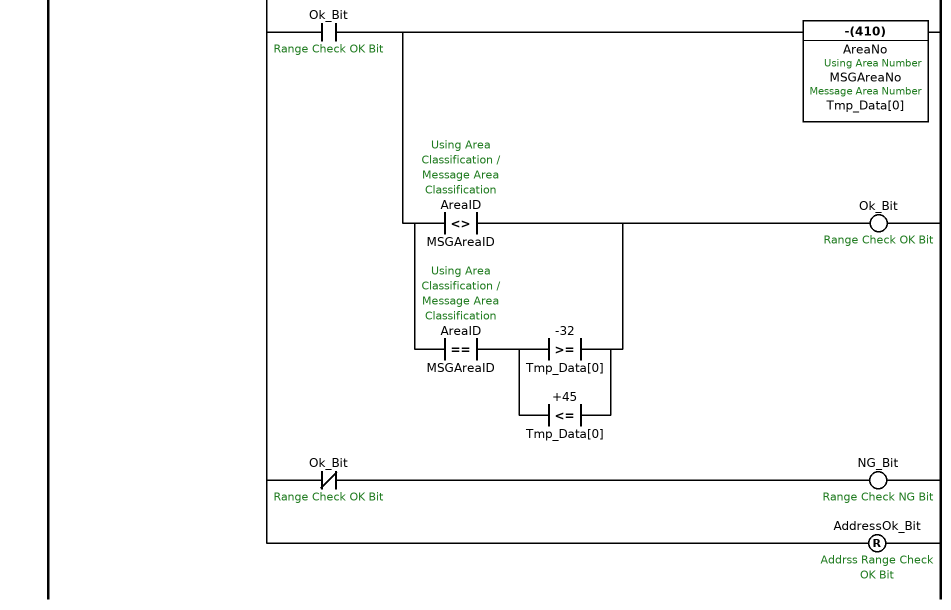
; [picture p24: FB INV002_Refresh_X31_, rungs 2-2]
; rung 2: Check input data range
LD EN
ANDNOT BUSY_Run  ; Internal Processing Flag
OR Data_Change  ; Detect input data change
OUT TR0
LD>=(325) &15 UnitSelect  ; Specify the connetcted Unit SCB=#BBBB_SCU=&0to&15
OR=(300) #BBBB UnitSelect  ; Specify the connetcted Unit SCB=#BBBB_SCU=&0to&15
OR=(300) #CCCC UnitSelect  ; Specify the connetcted Unit SCB=#BBBB_SCU=&0to&15
ANDLD
OUT Ok_Bit  ; Range Check OK Bit
LD TR0
AND Ok_Bit  ; Range Check OK Bit
AND<=(315) &1 PortNo  ; Serial port No. &0to&2
AND>=(325) &2 PortNo  ; Serial port No. &0to&2
OUT Ok_Bit  ; Range Check OK Bit
LD TR0
+(400) #4F P_EM_MaxNo EM_NoCheck  ; EM bank size, EM bank size check area
MOV(021) &62 Tmp_Data[0]
AND Ok_Bit  ; Range Check OK Bit
OUT TR1
AND=(300) #B0 AreaID  ; Using Area Classification
-(410) &6144 Tmp_Data[0] Tmp_Data[1]
AND>(320) Tmp_Data[1] AreaNo  ; Using Area Number
OUT Ok_IO  ; Selected CIO area range OK
LD TR1
AND=(300) #B1 AreaID  ; Using Area Classification
-(410) &512 Tmp_Data[0] Tmp_Data[1]
AND>(320) Tmp_Data[1] AreaNo  ; Using Area Number
OUT Ok_WR  ; Selected WR area range OK
LD TR1
AND=(300) #B2 AreaID  ; Using Area Classification
-(410) &512 Tmp_Data[0] Tmp_Data[1]
AND>(320) Tmp_Data[1] AreaNo  ; Using Area Number
OUT Ok_HR  ; Selected HR area range OK
LD TR1
AND=(300) #82 AreaID  ; Using Area Classification
-(410) &32768 Tmp_Data[0] Tmp_Data[1]
AND>(320) Tmp_Data[1] AreaNo  ; Using Area Number
OUT Ok_DM  ; Selected DM area range OK
LD TR1
AND<=(315) #50 AreaID  ; Using Area Classification
AND>=(325) EM_NoCheck AreaID  ; EM bank size check area, Using Area Classification
-(410) &32768 Tmp_Data[0] Tmp_Data[1]
AND>(320) Tmp_Data[1] AreaNo  ; Using Area Number
OUT Ok_EM  ; Selected EM area range OK
LD TR0
LD Ok_IO  ; Selected CIO area range OK
OR Ok_WR  ; Selected WR area range OK
OR Ok_HR  ; Selected HR area range OK
OR Ok_DM  ; Selected DM area range OK
OR Ok_EM  ; Selected EM area range OK
ANDLD
OUT Ok_Bit  ; Range Check OK Bit
LD TR0
MOV(021) &45 Tmp_Data[0]
AND Ok_Bit  ; Range Check OK Bit
OUT TR2
AND=(300) #B0 MSGAreaID  ; Message Area Classification
-(410) &6144 Tmp_Data[0] Tmp_Data[1]
AND>(320) Tmp_Data[1] MSGAreaNo  ; Message Area Number
OUT Ok_IO  ; Selected CIO area range OK
LD TR2
AND=(300) #B1 MSGAreaID  ; Message Area Classification
-(410) &512 Tmp_Data[0] Tmp_Data[1]
AND>(320) Tmp_Data[1] MSGAreaNo  ; Message Area Number
OUT Ok_WR  ; Selected WR area range OK
LD TR2
AND=(300) #B2 MSGAreaID  ; Message Area Classification
-(410) &512 Tmp_Data[0] Tmp_Data[1]
AND>(320) Tmp_Data[1] MSGAreaNo  ; Message Area Number
OUT Ok_HR  ; Selected HR area range OK
LD TR2
AND=(300) #82 MSGAreaID  ; Message Area Classification
-(410) &32768 Tmp_Data[0] Tmp_Data[1]
AND>(320) Tmp_Data[1] MSGAreaNo  ; Message Area Number
OUT Ok_DM  ; Selected DM area range OK
LD TR2
AND<=(315) #50 MSGAreaID  ; Message Area Classification
AND>=(325) EM_NoCheck MSGAreaID  ; EM bank size check area, Message Area Classification
-(410) &32768 Tmp_Data[0] Tmp_Data[1]
AND>(320) Tmp_Data[1] MSGAreaNo  ; Message Area Number
OUT Ok_EM  ; Selected EM area range OK
LD TR0
LD Ok_IO  ; Selected CIO area range OK
OR Ok_WR  ; Selected WR area range OK
OR Ok_HR  ; Selected HR area range OK
OR Ok_DM  ; Selected DM area range OK
OR Ok_EM  ; Selected EM area range OK
ANDLD
OUT Ok_Bit  ; Range Check OK Bit
LD TR0
AND Ok_Bit  ; Range Check OK Bit
-(410) AreaNo MSGAreaNo Tmp_Data[0]  ; Using Area Number, Message Area Number
LD<>(305) AreaID MSGAreaID  ; Using Area Classification, Message Area Classification
LD=(300) AreaID MSGAreaID  ; Using Area Classification, Message Area Classification
LD>=S(327) -32 Tmp_Data[0]
OR<=S(317) +45 Tmp_Data[0]
ANDLD
ORLD
ANDLD
OUT Ok_Bit  ; Range Check OK Bit
LD TR0
ANDNOT Ok_Bit  ; Range Check OK Bit
OUT NG_Bit  ; Range Check NG Bit
LD TR0
RSET AddressOk_Bit  ; Addrss Range Check OK Bit

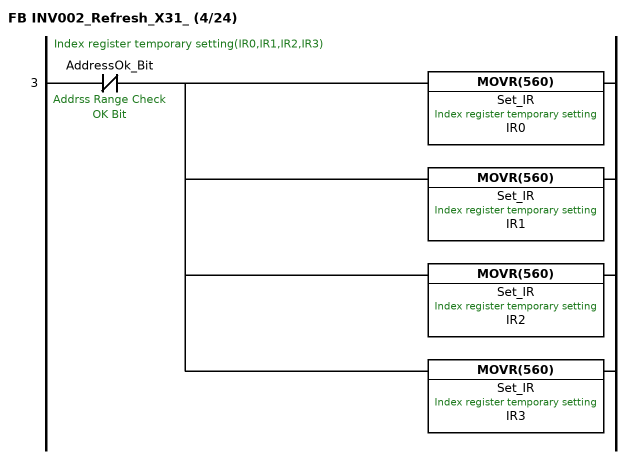
; rung 3: Index register temporary setting(IR0,IR1,IR2,IR3)
LDNOT AddressOk_Bit  ; Addrss Range Check OK Bit
MOVR(560) Set_IR IR0  ; Index register temporary setting
MOVR(560) Set_IR IR1  ; Index register temporary setting
MOVR(560) Set_IR IR2  ; Index register temporary setting
MOVR(560) Set_IR IR3  ; Index register temporary setting

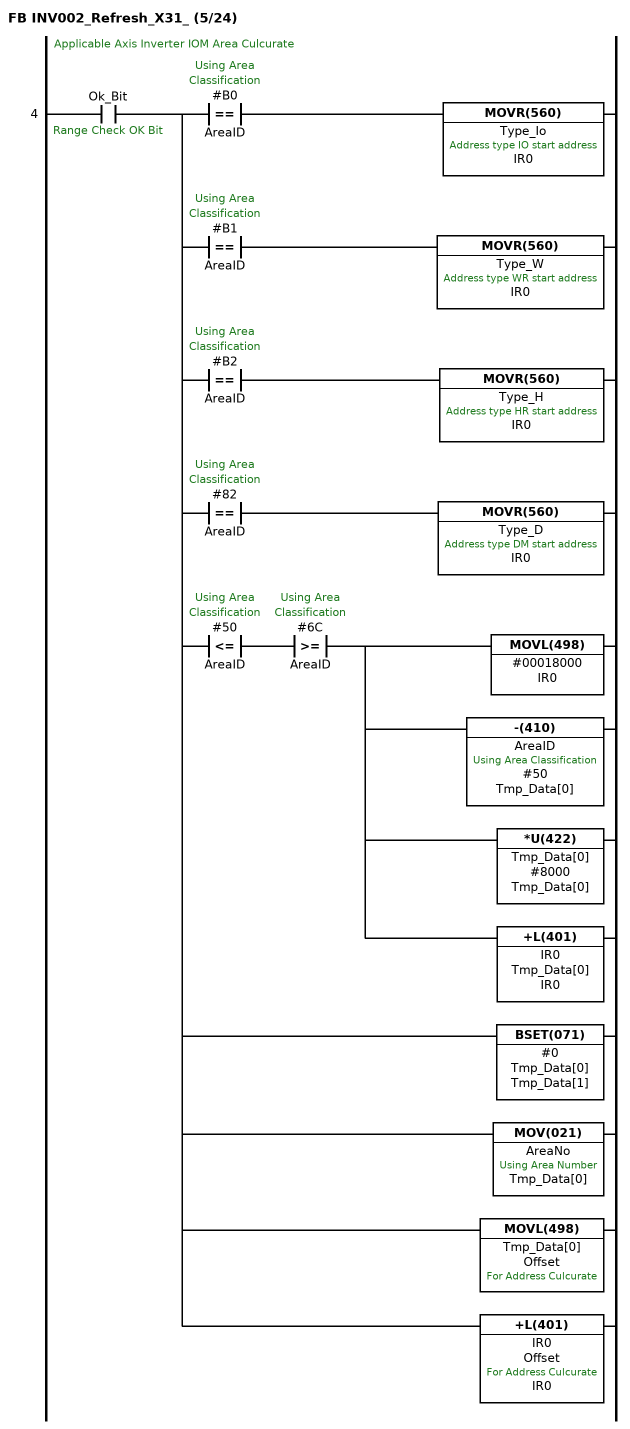
; rung 4: Applicable Axis Inverter IOM Area Culcurate
LD Ok_Bit  ; Range Check OK Bit
OUT TR0
AND=(300) #B0 AreaID  ; Using Area Classification
MOVR(560) Type_Io IR0  ; Address type IO start address
LD TR0
AND=(300) #B1 AreaID  ; Using Area Classification
MOVR(560) Type_W IR0  ; Address type WR start address
LD TR0
AND=(300) #B2 AreaID  ; Using Area Classification
MOVR(560) Type_H IR0  ; Address type HR start address
LD TR0
AND=(300) #82 AreaID  ; Using Area Classification
MOVR(560) Type_D IR0  ; Address type DM start address
LD TR0
AND<=(315) #50 AreaID  ; Using Area Classification
AND>=(325) #6C AreaID  ; Using Area Classification
MOVL(498) #00018000 IR0
-(410) AreaID #50 Tmp_Data[0]  ; Using Area Classification
*U(422) Tmp_Data[0] #8000 Tmp_Data[0]
+L(401) IR0 Tmp_Data[0] IR0
LD TR0
BSET(071) #0 Tmp_Data[0] Tmp_Data[1]
MOV(021) AreaNo Tmp_Data[0]  ; Using Area Number
MOVL(498) Tmp_Data[0] Offset  ; For Address Culcurate
+L(401) IR0 Offset IR0  ; For Address Culcurate

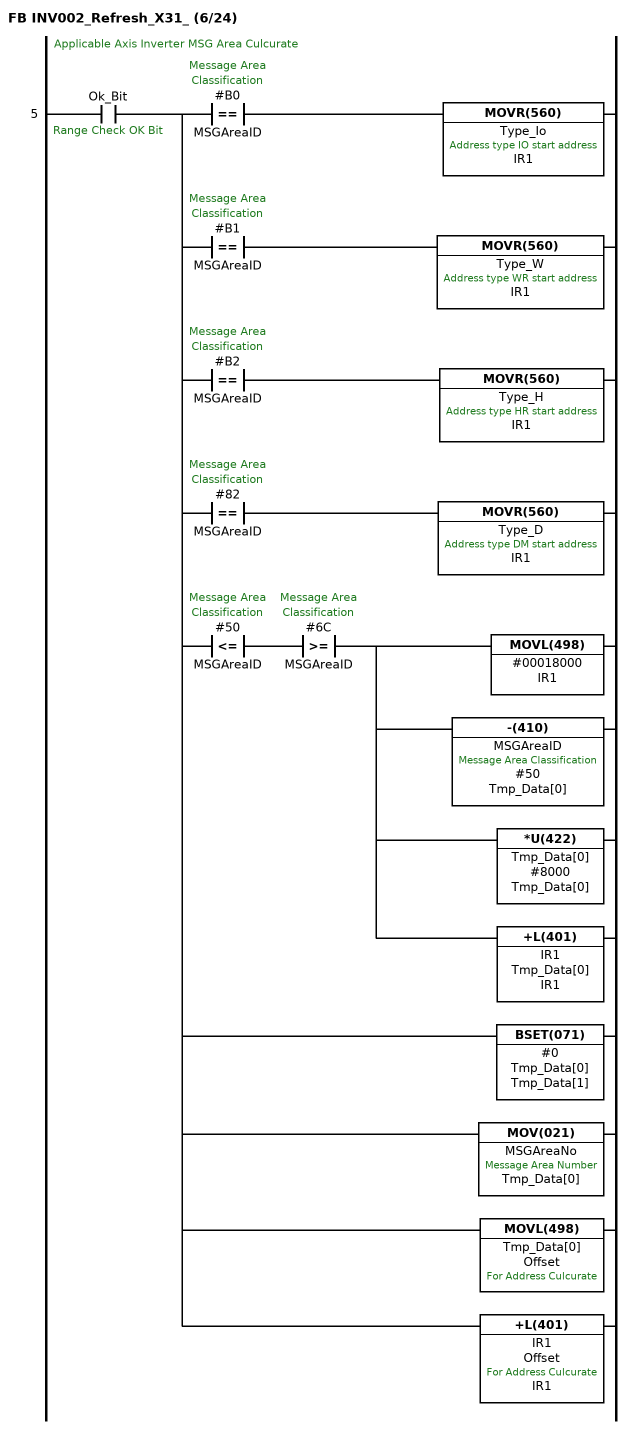
; rung 5: Applicable Axis Inverter MSG Area Culcurate
LD Ok_Bit  ; Range Check OK Bit
OUT TR0
AND=(300) #B0 MSGAreaID  ; Message Area Classification
MOVR(560) Type_Io IR1  ; Address type IO start address
LD TR0
AND=(300) #B1 MSGAreaID  ; Message Area Classification
MOVR(560) Type_W IR1  ; Address type WR start address
LD TR0
AND=(300) #B2 MSGAreaID  ; Message Area Classification
MOVR(560) Type_H IR1  ; Address type HR start address
LD TR0
AND=(300) #82 MSGAreaID  ; Message Area Classification
MOVR(560) Type_D IR1  ; Address type DM start address
LD TR0
AND<=(315) #50 MSGAreaID  ; Message Area Classification
AND>=(325) #6C MSGAreaID  ; Message Area Classification
MOVL(498) #00018000 IR1
-(410) MSGAreaID #50 Tmp_Data[0]  ; Message Area Classification
*U(422) Tmp_Data[0] #8000 Tmp_Data[0]
+L(401) IR1 Tmp_Data[0] IR1
LD TR0
BSET(071) #0 Tmp_Data[0] Tmp_Data[1]
MOV(021) MSGAreaNo Tmp_Data[0]  ; Message Area Number
MOVL(498) Tmp_Data[0] Offset  ; For Address Culcurate
+L(401) IR1 Offset IR1  ; For Address Culcurate

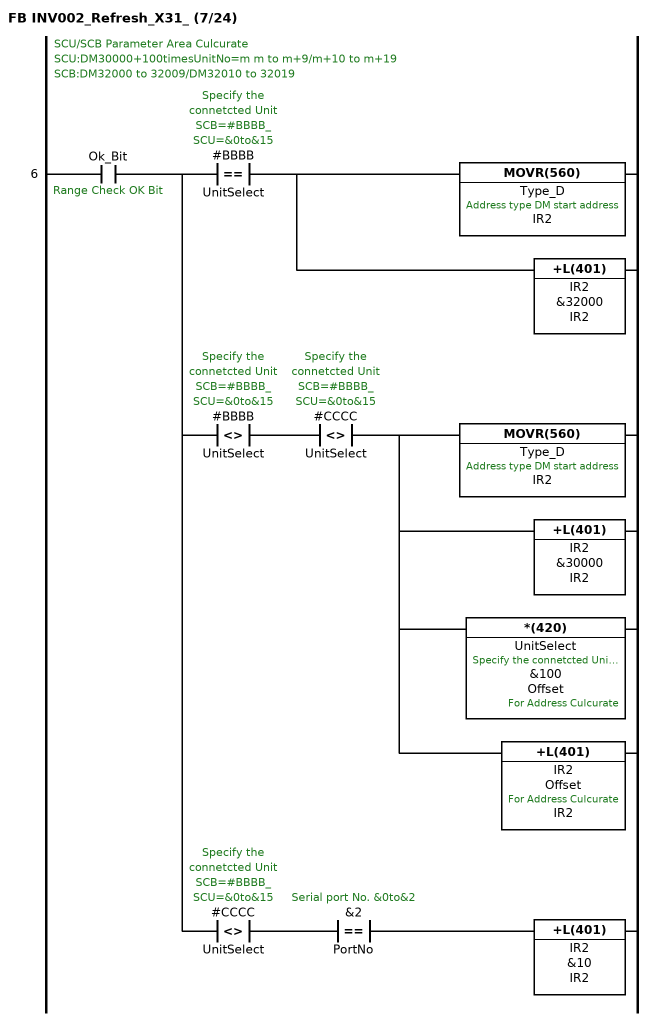
; rung 6: SCU/SCB Parameter Area Culcurate / SCU:DM30000+100timesUnitNo=m m to m+9/m+10 to m+19 / SCB:DM32000 to 32009/DM32010 to 32019
LD Ok_Bit  ; Range Check OK Bit
OUT TR0
AND=(300) #BBBB UnitSelect  ; Specify the connetcted Unit SCB=#BBBB_SCU=&0to&15
MOVR(560) Type_D IR2  ; Address type DM start address
+L(401) IR2 &32000 IR2
LD TR0
AND<>(305) #BBBB UnitSelect  ; Specify the connetcted Unit SCB=#BBBB_SCU=&0to&15
AND<>(305) #CCCC UnitSelect  ; Specify the connetcted Unit SCB=#BBBB_SCU=&0to&15
MOVR(560) Type_D IR2  ; Address type DM start address
+L(401) IR2 &30000 IR2
*(420) UnitSelect &100 Offset  ; Specify the connetcted Unit SCB=#BBBB_SCU=&0to&15, For Address Culcurate
+L(401) IR2 Offset IR2  ; For Address Culcurate
LD TR0
AND<>(305) #CCCC UnitSelect  ; Specify the connetcted Unit SCB=#BBBB_SCU=&0to&15
AND=(300) &2 PortNo  ; Serial port No. &0to&2
+L(401) IR2 &10 IR2

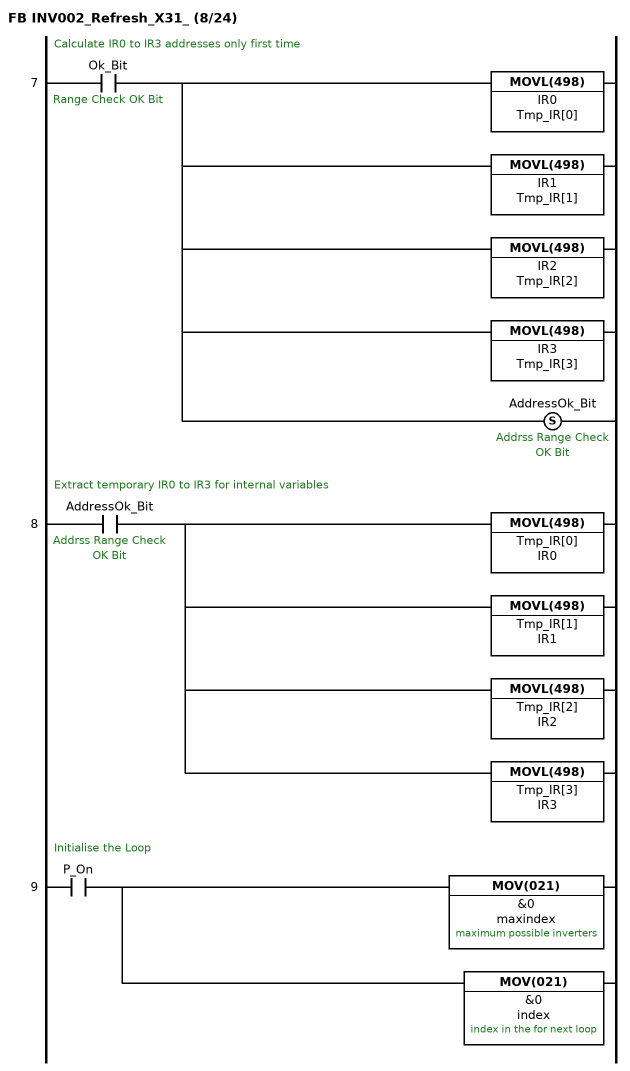
; rung 7: Calculate IR0 to IR3 addresses only first time
LD Ok_Bit  ; Range Check OK Bit
MOVL(498) IR0 Tmp_IR[0]
MOVL(498) IR1 Tmp_IR[1]
MOVL(498) IR2 Tmp_IR[2]
MOVL(498) IR3 Tmp_IR[3]
SET AddressOk_Bit  ; Addrss Range Check OK Bit
; rung 8: Extract temporary IR0 to IR3 for internal variables
LD AddressOk_Bit  ; Addrss Range Check OK Bit
MOVL(498) Tmp_IR[0] IR0
MOVL(498) Tmp_IR[1] IR1
MOVL(498) Tmp_IR[2] IR2
MOVL(498) Tmp_IR[3] IR3
; rung 9: Initialise the Loop
LD P_On
MOV(021) &0 maxindex  ; maximum possible inverters
MOV(021) &0 index  ; index in the for next loop

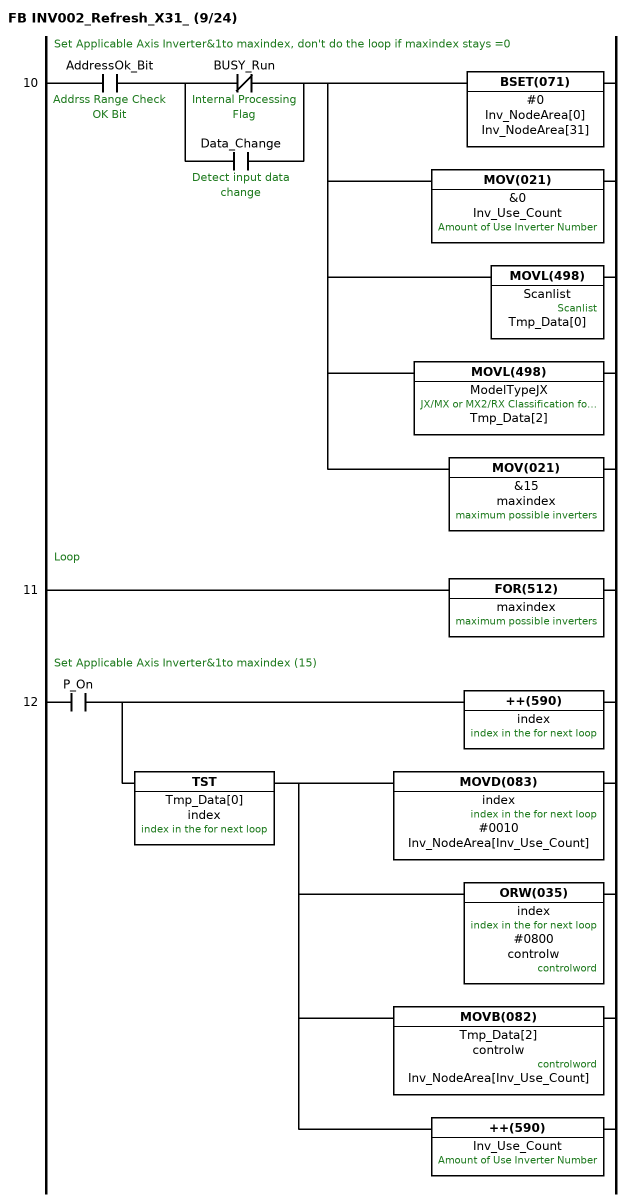
; rung 10: Set Applicable Axis Inverter&1to maxindex, don't do the loop if maxindex stays =0
LD AddressOk_Bit  ; Addrss Range Check OK Bit
LDNOT BUSY_Run  ; Internal Processing Flag
OR Data_Change  ; Detect input data change
ANDLD
BSET(071) #0 Inv_NodeArea[0] Inv_NodeArea[31]
MOV(021) &0 Inv_Use_Count  ; Amount of Use Inverter Number
MOVL(498) Scanlist Tmp_Data[0]  ; Scanlist
MOVL(498) ModelTypeJX Tmp_Data[2]  ; JX/MX or MX2/RX Classification for older Inverter types also this Bit has to be set, like scanlist
MOV(021) &15 maxindex  ; maximum possible inverters
; rung 11: Loop
FOR(512) maxindex  ; maximum possible inverters
; rung 12: Set Applicable Axis Inverter&1to maxindex (15)
LD P_On
++(590) index  ; index in the for next loop
ANDTST(350) Tmp_Data[0] index  ; index in the for next loop
MOVD(083) index #0010 Inv_NodeArea[Inv_Use_Count]  ; index in the for next loop
ORW(035) index #0800 controlw  ; index in the for next loop, controlword
MOVB(082) Tmp_Data[2] controlw Inv_NodeArea[Inv_Use_Count]  ; controlword
++(590) Inv_Use_Count  ; Amount of Use Inverter Number

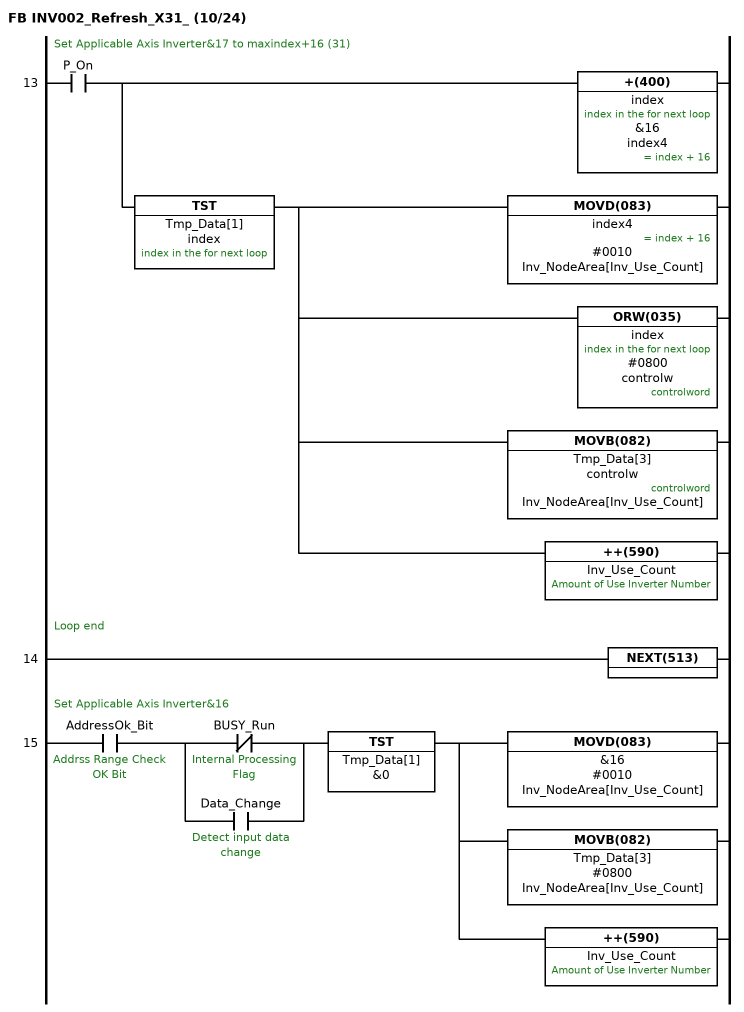
; rung 13: Set Applicable Axis Inverter&17 to maxindex+16 (31)
LD P_On
+(400) index &16 index4  ; index in the for next loop, = index + 16
ANDTST(350) Tmp_Data[1] index  ; index in the for next loop
MOVD(083) index4 #0010 Inv_NodeArea[Inv_Use_Count]  ; = index + 16
ORW(035) index #0800 controlw  ; index in the for next loop, controlword
MOVB(082) Tmp_Data[3] controlw Inv_NodeArea[Inv_Use_Count]  ; controlword
++(590) Inv_Use_Count  ; Amount of Use Inverter Number
; rung 14: Loop end
NEXT(513)
; rung 15: Set Applicable Axis Inverter&16
LD AddressOk_Bit  ; Addrss Range Check OK Bit
LDNOT BUSY_Run  ; Internal Processing Flag
OR Data_Change  ; Detect input data change
ANDLD
ANDTST(350) Tmp_Data[1] &0
MOVD(083) &16 #0010 Inv_NodeArea[Inv_Use_Count]
MOVB(082) Tmp_Data[3] #0800 Inv_NodeArea[Inv_Use_Count]
++(590) Inv_Use_Count  ; Amount of Use Inverter Number

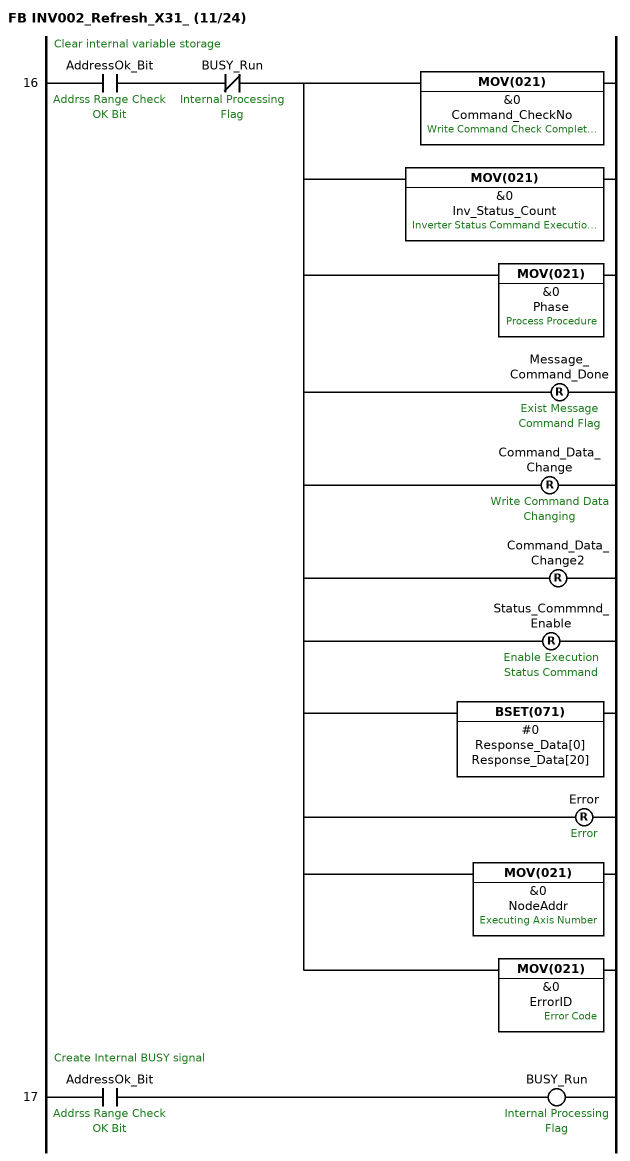
; rung 16: Clear internal variable storage
LD AddressOk_Bit  ; Addrss Range Check OK Bit
ANDNOT BUSY_Run  ; Internal Processing Flag
MOV(021) &0 Command_CheckNo  ; Write Command Check Complete Number
MOV(021) &0 Inv_Status_Count  ; Inverter Status Command Execution Number
MOV(021) &0 Phase  ; Process Procedure
RSET Message_Command_Done  ; Exist Message Command Flag
RSET Command_Data_Change  ; Write Command Data Changing
RSET Command_Data_Change2
RSET Status_Commmnd_Enable  ; Enable Execution Status Command
BSET(071) #0 Response_Data[0] Response_Data[20]
RSET Error  ; Error
MOV(021) &0 NodeAddr  ; Executing Axis Number
MOV(021) &0 ErrorID  ; Error Code
; rung 17: Create Internal BUSY signal
LD AddressOk_Bit  ; Addrss Range Check OK Bit
OUT BUSY_Run  ; Internal Processing Flag

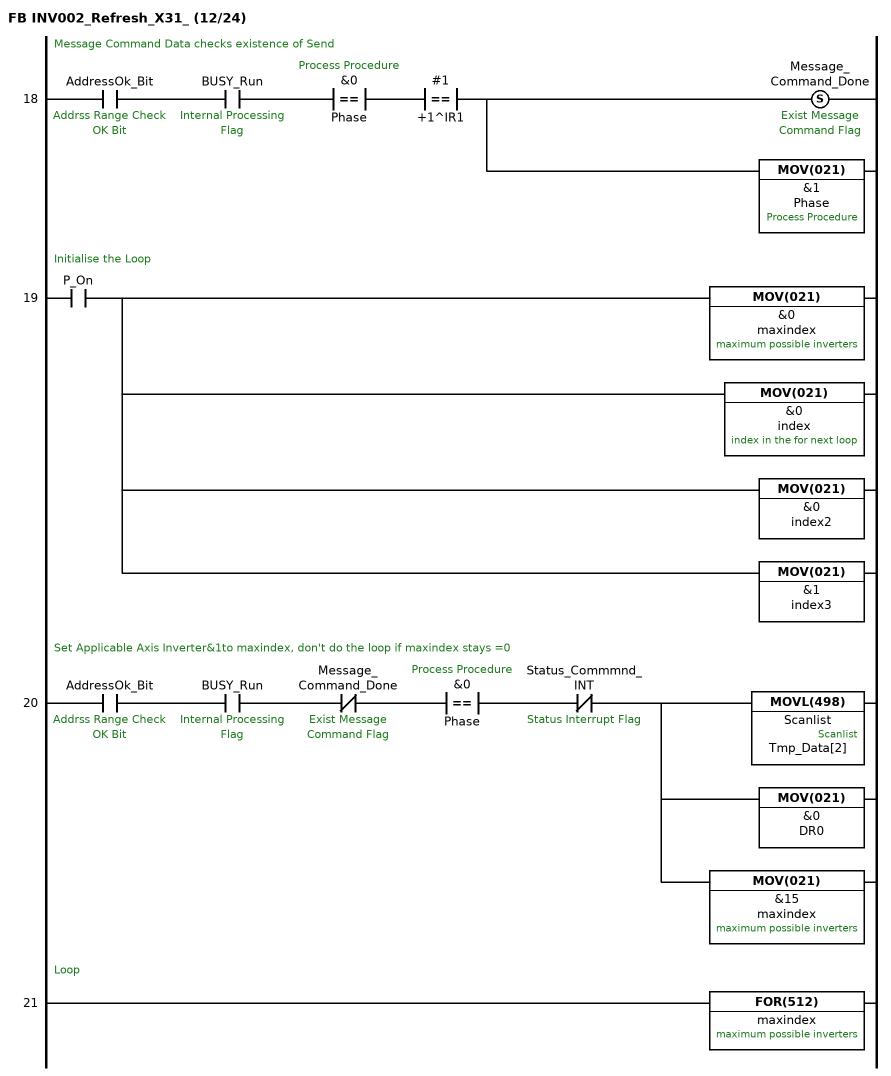
; rung 18: Message Command Data checks existence of Send
LD AddressOk_Bit  ; Addrss Range Check OK Bit
AND BUSY_Run  ; Internal Processing Flag
AND=(300) &0 Phase  ; Process Procedure
AND=(300) #1 +1^IR1
SET Message_Command_Done  ; Exist Message Command Flag
MOV(021) &1 Phase  ; Process Procedure
; rung 19: Initialise the Loop
LD P_On
MOV(021) &0 maxindex  ; maximum possible inverters
MOV(021) &0 index  ; index in the for next loop
MOV(021) &0 index2
MOV(021) &1 index3
; rung 20: Set Applicable Axis Inverter&1to maxindex, don't do the loop if maxindex stays =0
LD AddressOk_Bit  ; Addrss Range Check OK Bit
AND BUSY_Run  ; Internal Processing Flag
ANDNOT Message_Command_Done  ; Exist Message Command Flag
AND=(300) &0 Phase  ; Process Procedure
ANDNOT Status_Commmnd_INT  ; Status Interrupt Flag
MOVL(498) Scanlist Tmp_Data[2]  ; Scanlist
MOV(021) &0 DR0
MOV(021) &15 maxindex  ; maximum possible inverters
; rung 21: Loop
FOR(512) maxindex  ; maximum possible inverters

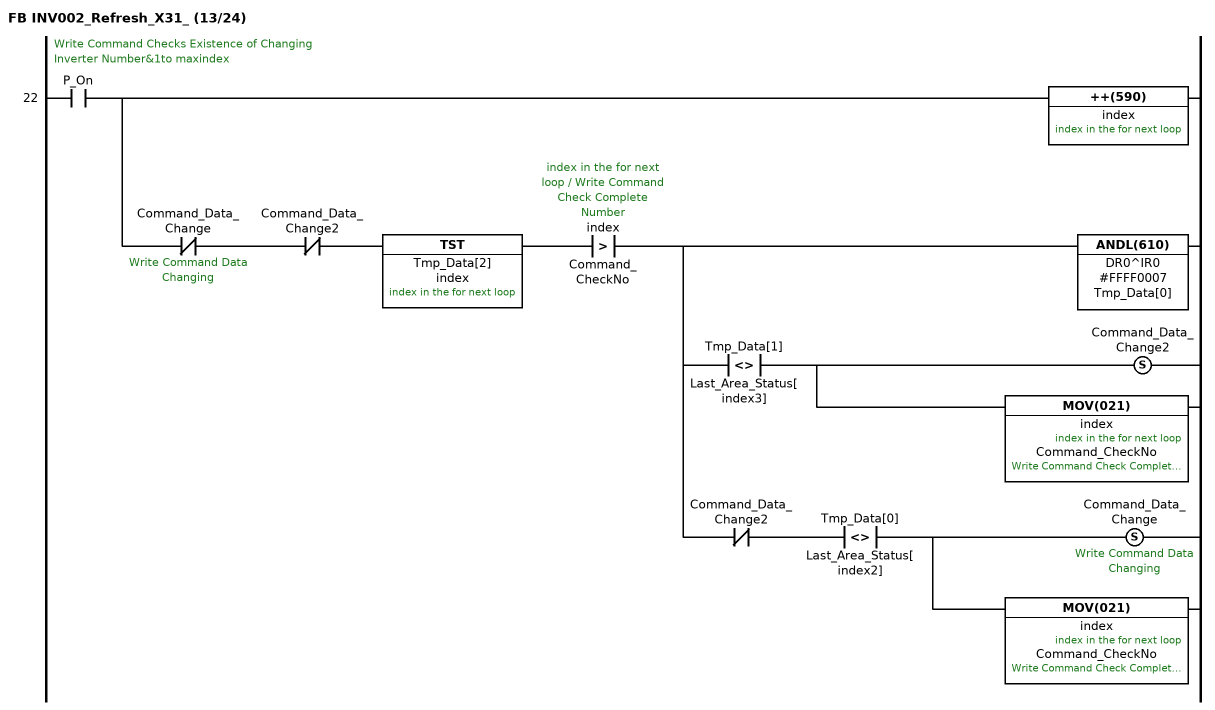
; rung 22: Write Command Checks Existence of Changing / Inverter Number&1to maxindex
LD P_On
++(590) index  ; index in the for next loop
ANDNOT Command_Data_Change  ; Write Command Data Changing
ANDNOT Command_Data_Change2
ANDTST(350) Tmp_Data[2] index  ; index in the for next loop
AND>(320) index Command_CheckNo  ; index in the for next loop, Write Command Check Complete Number
OUT TR0
ANDL(610) DR0^IR0 #FFFF0007 Tmp_Data[0]
AND<>(305) Tmp_Data[1] Last_Area_Status[index3]
SET Command_Data_Change2
MOV(021) index Command_CheckNo  ; index in the for next loop, Write Command Check Complete Number
LD TR0
ANDNOT Command_Data_Change2
AND<>(305) Tmp_Data[0] Last_Area_Status[index2]
SET Command_Data_Change  ; Write Command Data Changing
MOV(021) index Command_CheckNo  ; index in the for next loop, Write Command Check Complete Number

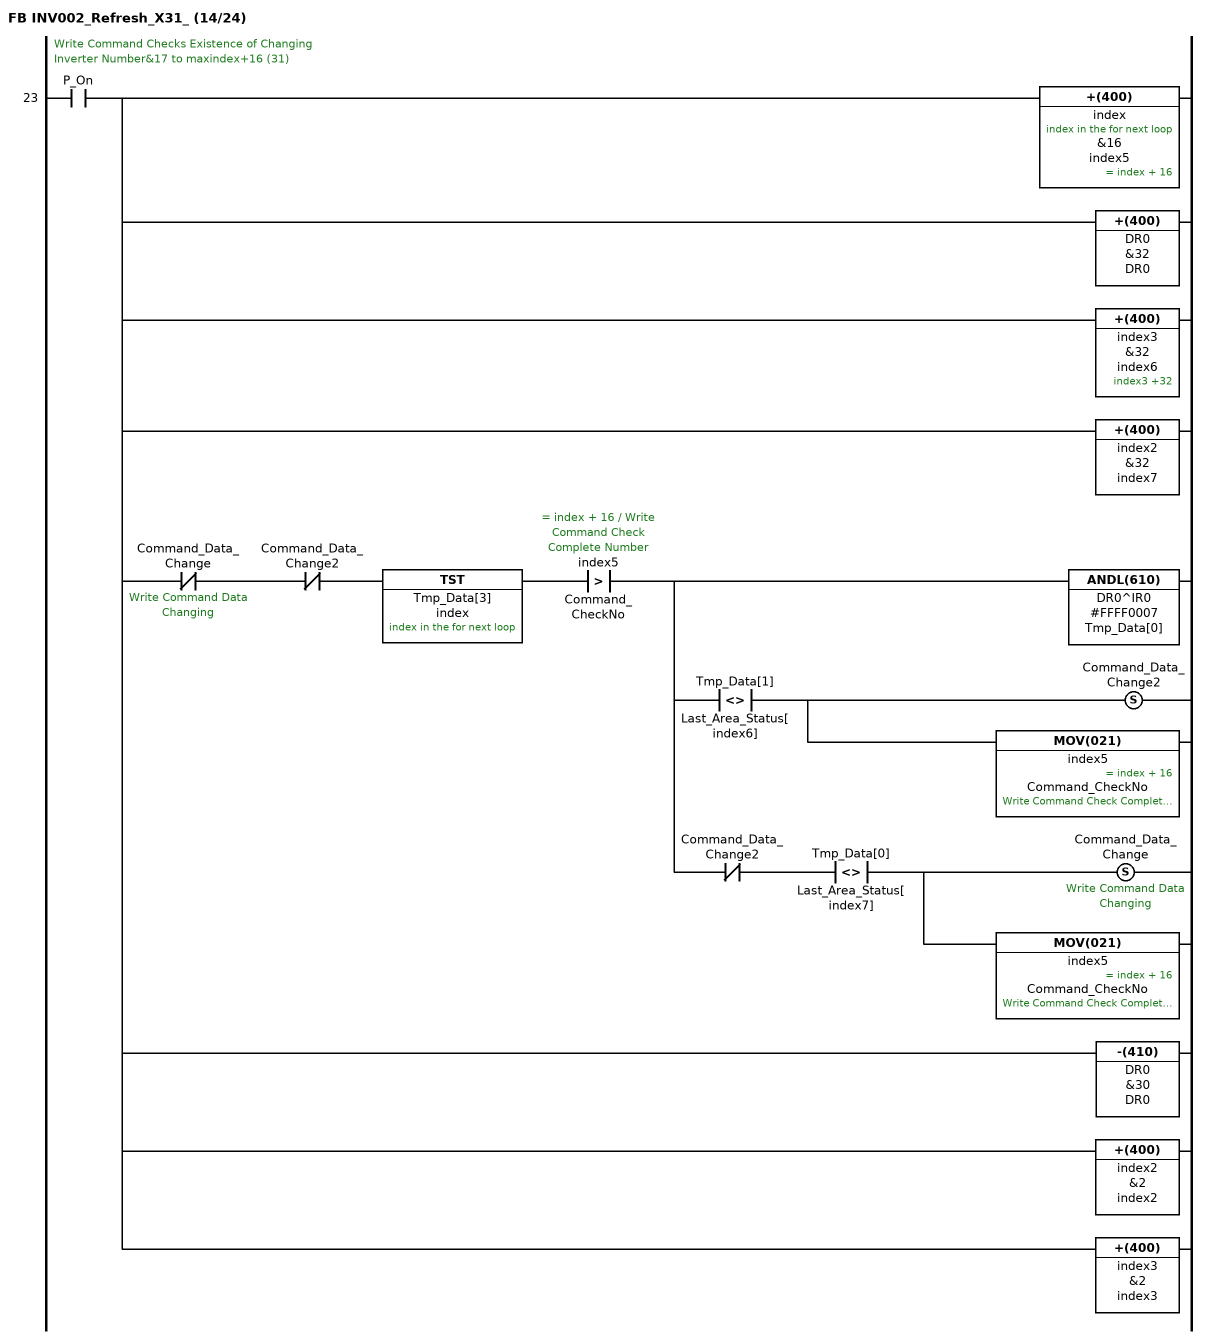
; rung 23: Write Command Checks Existence of Changing / Inverter Number&17 to maxindex+16 (31)
LD P_On
OUT TR0
+(400) index &16 index5  ; index in the for next loop, = index + 16
+(400) DR0 &32 DR0
+(400) index3 &32 index6  ; index3 +32
+(400) index2 &32 index7
ANDNOT Command_Data_Change  ; Write Command Data Changing
ANDNOT Command_Data_Change2
ANDTST(350) Tmp_Data[3] index  ; index in the for next loop
AND>(320) index5 Command_CheckNo  ; = index + 16, Write Command Check Complete Number
OUT TR1
ANDL(610) DR0^IR0 #FFFF0007 Tmp_Data[0]
AND<>(305) Tmp_Data[1] Last_Area_Status[index6]
SET Command_Data_Change2
MOV(021) index5 Command_CheckNo  ; = index + 16, Write Command Check Complete Number
LD TR1
ANDNOT Command_Data_Change2
AND<>(305) Tmp_Data[0] Last_Area_Status[index7]
SET Command_Data_Change  ; Write Command Data Changing
MOV(021) index5 Command_CheckNo  ; = index + 16, Write Command Check Complete Number
LD TR0
-(410) DR0 &30 DR0
+(400) index2 &2 index2
+(400) index3 &2 index3

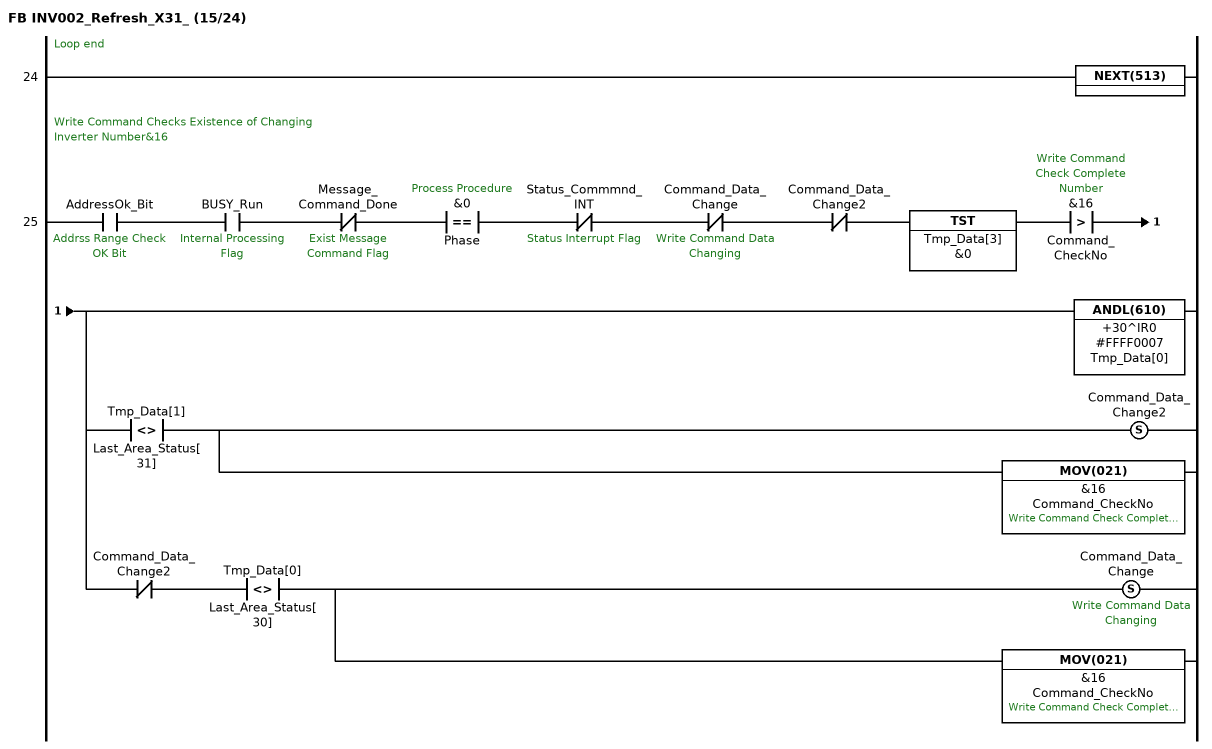
; rung 24: Loop end
NEXT(513)
; rung 25: Write Command Checks Existence of Changing / Inverter Number&16
LD AddressOk_Bit  ; Addrss Range Check OK Bit
AND BUSY_Run  ; Internal Processing Flag
ANDNOT Message_Command_Done  ; Exist Message Command Flag
AND=(300) &0 Phase  ; Process Procedure
ANDNOT Status_Commmnd_INT  ; Status Interrupt Flag
ANDNOT Command_Data_Change  ; Write Command Data Changing
ANDNOT Command_Data_Change2
ANDTST(350) Tmp_Data[3] &0
AND>(320) &16 Command_CheckNo  ; Write Command Check Complete Number
OUT TR0
ANDL(610) +30^IR0 #FFFF0007 Tmp_Data[0]
AND<>(305) Tmp_Data[1] Last_Area_Status[31]
SET Command_Data_Change2
MOV(021) &16 Command_CheckNo  ; Write Command Check Complete Number
LD TR0
ANDNOT Command_Data_Change2
AND<>(305) Tmp_Data[0] Last_Area_Status[30]
SET Command_Data_Change  ; Write Command Data Changing
MOV(021) &16 Command_CheckNo  ; Write Command Check Complete Number

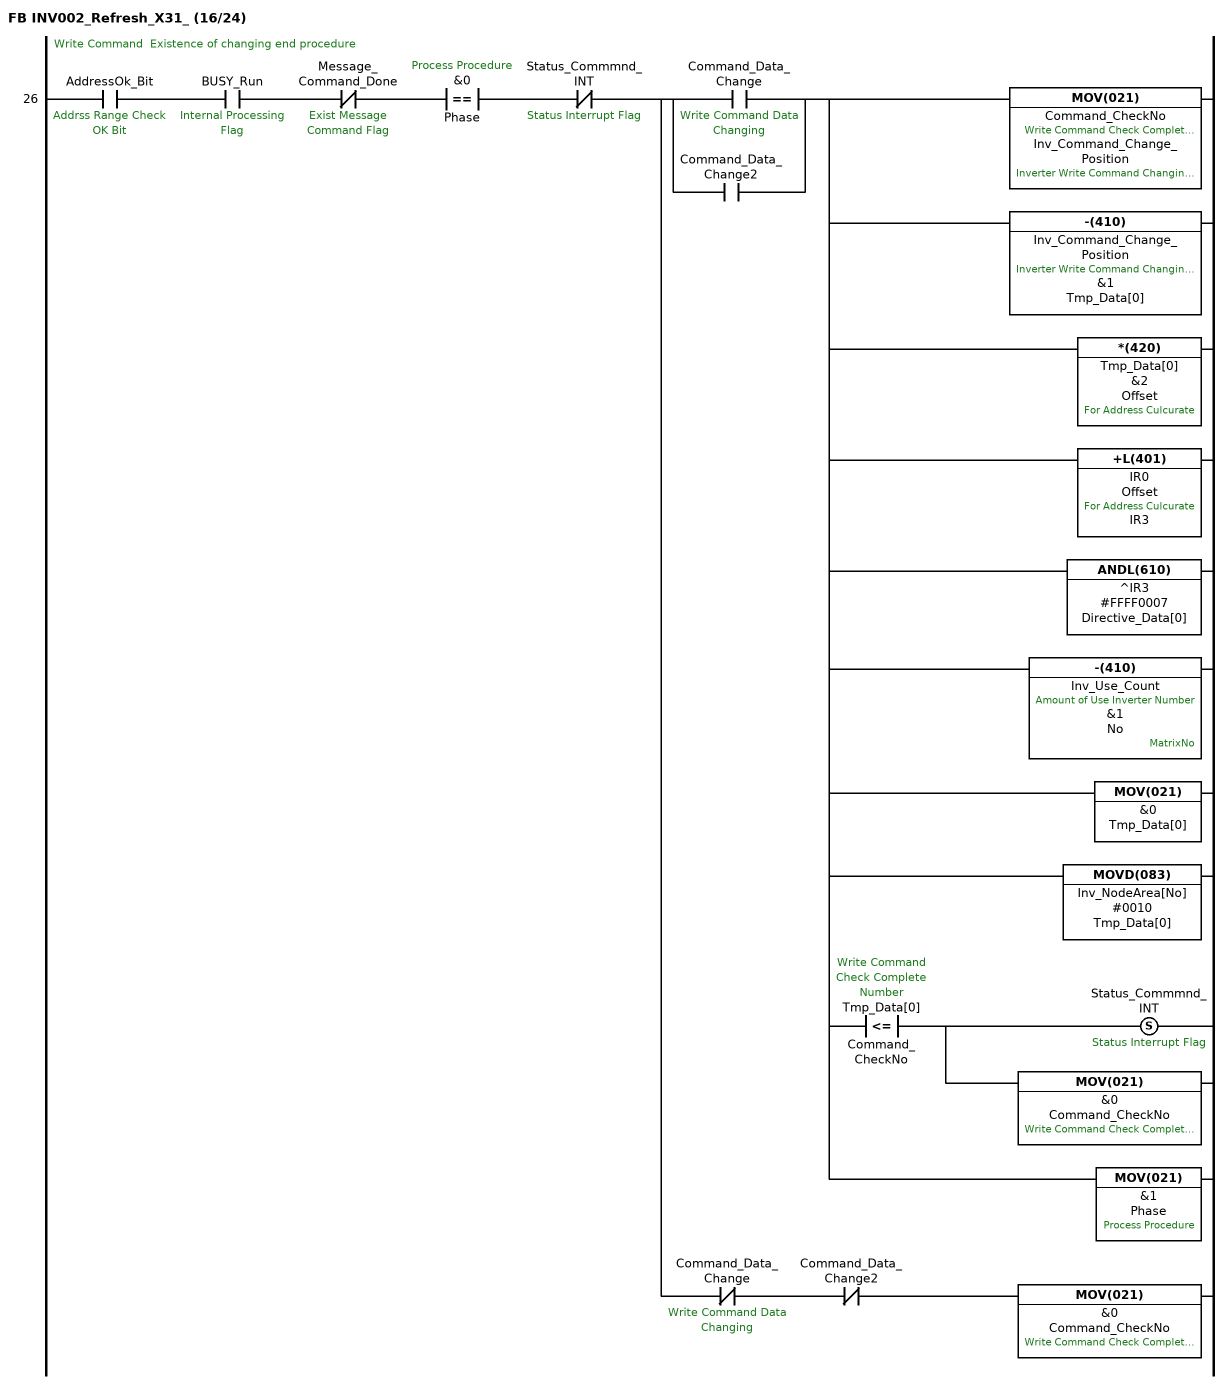
; rung 26: Write Command  Existence of changing end procedure
LD AddressOk_Bit  ; Addrss Range Check OK Bit
AND BUSY_Run  ; Internal Processing Flag
ANDNOT Message_Command_Done  ; Exist Message Command Flag
AND=(300) &0 Phase  ; Process Procedure
ANDNOT Status_Commmnd_INT  ; Status Interrupt Flag
OUT TR0
LD Command_Data_Change  ; Write Command Data Changing
OR Command_Data_Change2
ANDLD
OUT TR1
MOV(021) Command_CheckNo Inv_Command_Change_Position  ; Write Command Check Complete Number, Inverter Write Command Changing Position
-(410) Inv_Command_Change_Position &1 Tmp_Data[0]  ; Inverter Write Command Changing Position
*(420) Tmp_Data[0] &2 Offset  ; For Address Culcurate
+L(401) IR0 Offset IR3  ; For Address Culcurate
ANDL(610) ^IR3 #FFFF0007 Directive_Data[0]
-(410) Inv_Use_Count &1 No  ; Amount of Use Inverter Number, MatrixNo
MOV(021) &0 Tmp_Data[0]
MOVD(083) Inv_NodeArea[No] #0010 Tmp_Data[0]
AND<=(315) Tmp_Data[0] Command_CheckNo  ; Write Command Check Complete Number
SET Status_Commmnd_INT  ; Status Interrupt Flag
MOV(021) &0 Command_CheckNo  ; Write Command Check Complete Number
LD TR1
MOV(021) &1 Phase  ; Process Procedure
LD TR0
ANDNOT Command_Data_Change  ; Write Command Data Changing
ANDNOT Command_Data_Change2
MOV(021) &0 Command_CheckNo  ; Write Command Check Complete Number

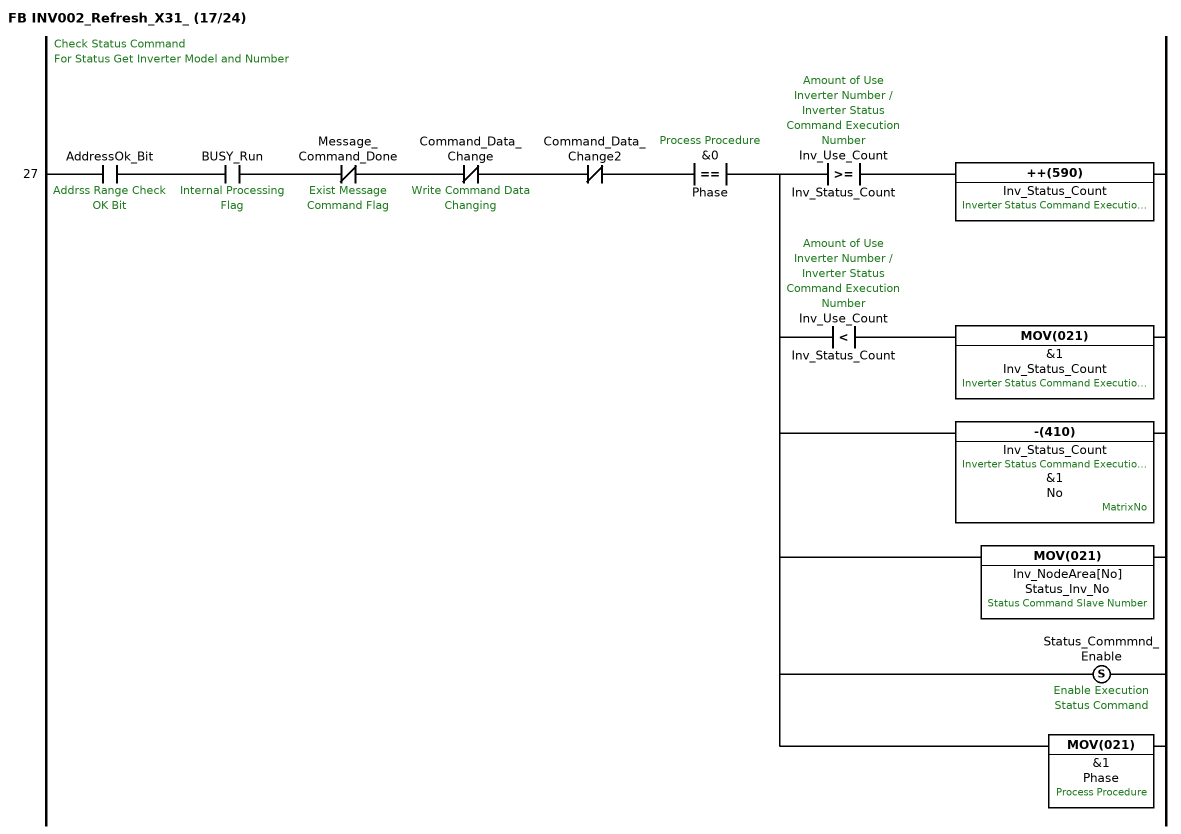
; rung 27: Check Status Command / For Status Get Inverter Model and Number
LD AddressOk_Bit  ; Addrss Range Check OK Bit
AND BUSY_Run  ; Internal Processing Flag
ANDNOT Message_Command_Done  ; Exist Message Command Flag
ANDNOT Command_Data_Change  ; Write Command Data Changing
ANDNOT Command_Data_Change2
AND=(300) &0 Phase  ; Process Procedure
OUT TR0
AND>=(325) Inv_Use_Count Inv_Status_Count  ; Amount of Use Inverter Number, Inverter Status Command Execution Number
++(590) Inv_Status_Count  ; Inverter Status Command Execution Number
LD TR0
AND<(310) Inv_Use_Count Inv_Status_Count  ; Amount of Use Inverter Number, Inverter Status Command Execution Number
MOV(021) &1 Inv_Status_Count  ; Inverter Status Command Execution Number
LD TR0
-(410) Inv_Status_Count &1 No  ; Inverter Status Command Execution Number, MatrixNo
MOV(021) Inv_NodeArea[No] Status_Inv_No  ; Status Command Slave Number
SET Status_Commmnd_Enable  ; Enable Execution Status Command
MOV(021) &1 Phase  ; Process Procedure

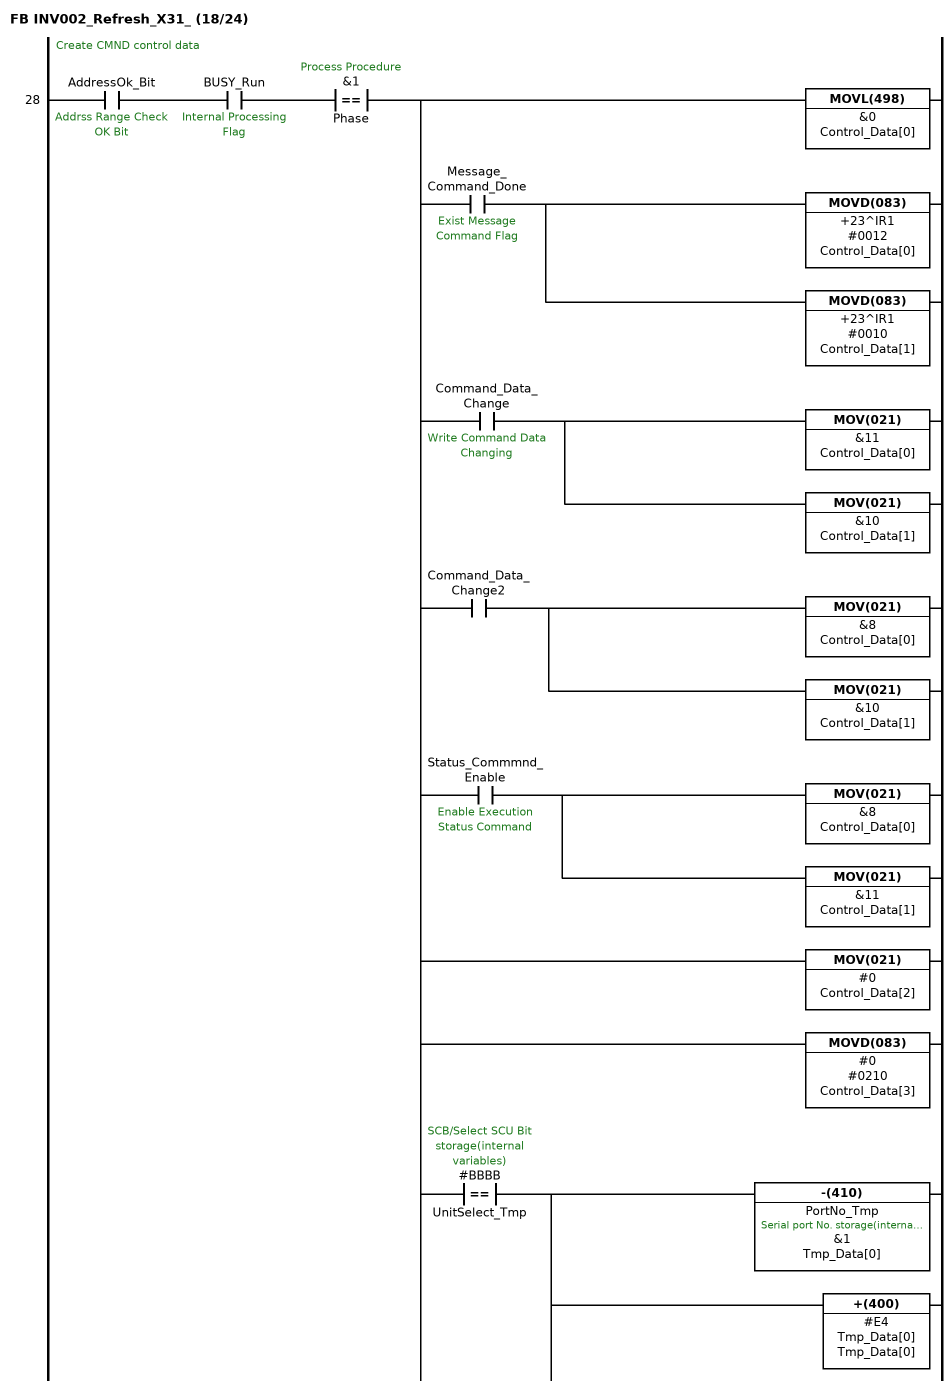

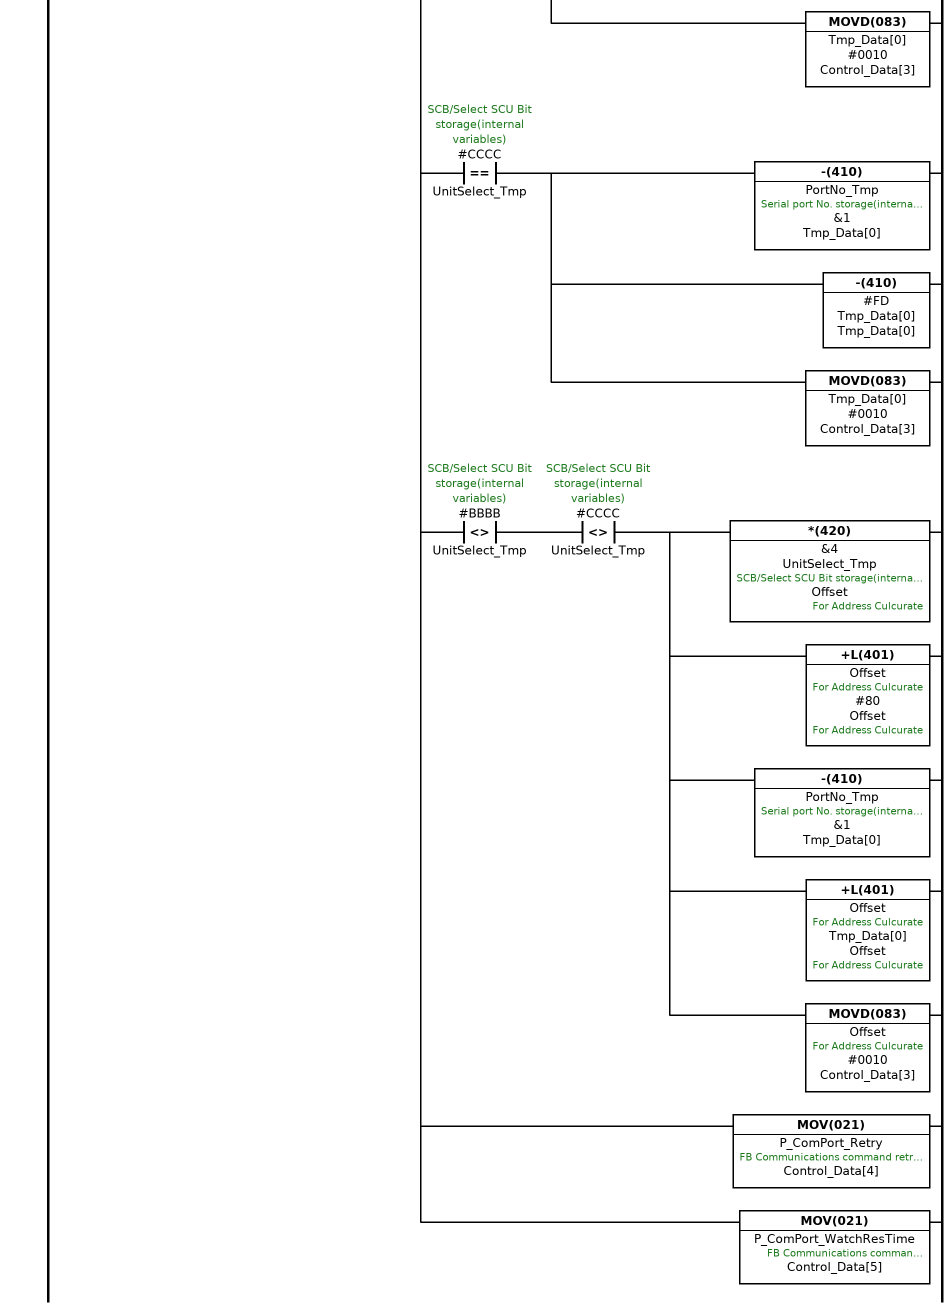
; rung 28: Create CMND control data
LD AddressOk_Bit  ; Addrss Range Check OK Bit
AND BUSY_Run  ; Internal Processing Flag
AND=(300) &1 Phase  ; Process Procedure
OUT TR0
MOVL(498) &0 Control_Data[0]
AND Message_Command_Done  ; Exist Message Command Flag
MOVD(083) +23^IR1 #0012 Control_Data[0]
MOVD(083) +23^IR1 #0010 Control_Data[1]
LD TR0
AND Command_Data_Change  ; Write Command Data Changing
MOV(021) &11 Control_Data[0]
MOV(021) &10 Control_Data[1]
LD TR0
AND Command_Data_Change2
MOV(021) &8 Control_Data[0]
MOV(021) &10 Control_Data[1]
LD TR0
AND Status_Commmnd_Enable  ; Enable Execution Status Command
MOV(021) &8 Control_Data[0]
MOV(021) &11 Control_Data[1]
LD TR0
MOV(021) #0 Control_Data[2]
MOVD(083) #0 #0210 Control_Data[3]
AND=(300) #BBBB UnitSelect_Tmp  ; SCB/Select SCU Bit storage(internal variables)
-(410) PortNo_Tmp &1 Tmp_Data[0]  ; Serial port No. storage(internal variables)
+(400) #E4 Tmp_Data[0] Tmp_Data[0]
MOVD(083) Tmp_Data[0] #0010 Control_Data[3]
LD TR0
AND=(300) #CCCC UnitSelect_Tmp  ; SCB/Select SCU Bit storage(internal variables)
-(410) PortNo_Tmp &1 Tmp_Data[0]  ; Serial port No. storage(internal variables)
-(410) #FD Tmp_Data[0] Tmp_Data[0]
MOVD(083) Tmp_Data[0] #0010 Control_Data[3]
LD TR0
AND<>(305) #BBBB UnitSelect_Tmp  ; SCB/Select SCU Bit storage(internal variables)
AND<>(305) #CCCC UnitSelect_Tmp  ; SCB/Select SCU Bit storage(internal variables)
*(420) &4 UnitSelect_Tmp Offset  ; SCB/Select SCU Bit storage(internal variables), For Address Culcurate
+L(401) Offset #80 Offset  ; For Address Culcurate
-(410) PortNo_Tmp &1 Tmp_Data[0]  ; Serial port No. storage(internal variables)
+L(401) Offset Tmp_Data[0] Offset  ; For Address Culcurate
MOVD(083) Offset #0010 Control_Data[3]  ; For Address Culcurate
LD TR0
MOV(021) P_ComPort_Retry Control_Data[4]  ; FB Communications command retry count
MOV(021) P_ComPort_WatchResTime Control_Data[5]  ; FB Communications command response Monitor time

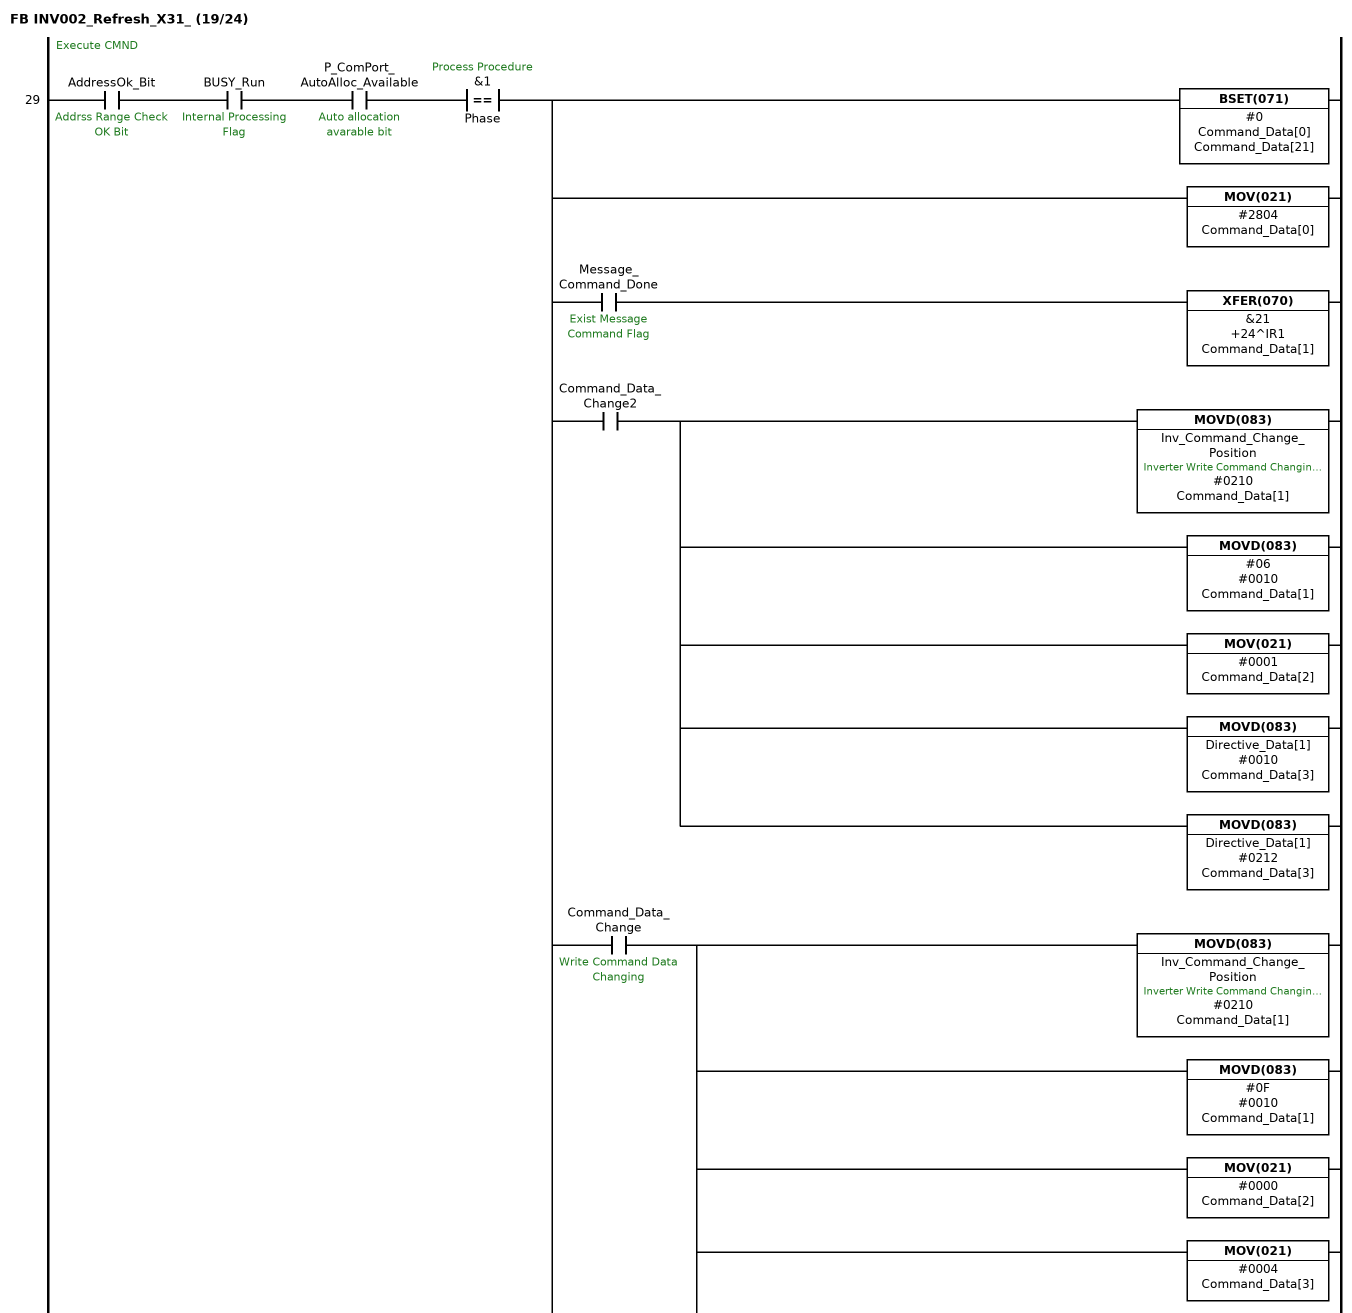

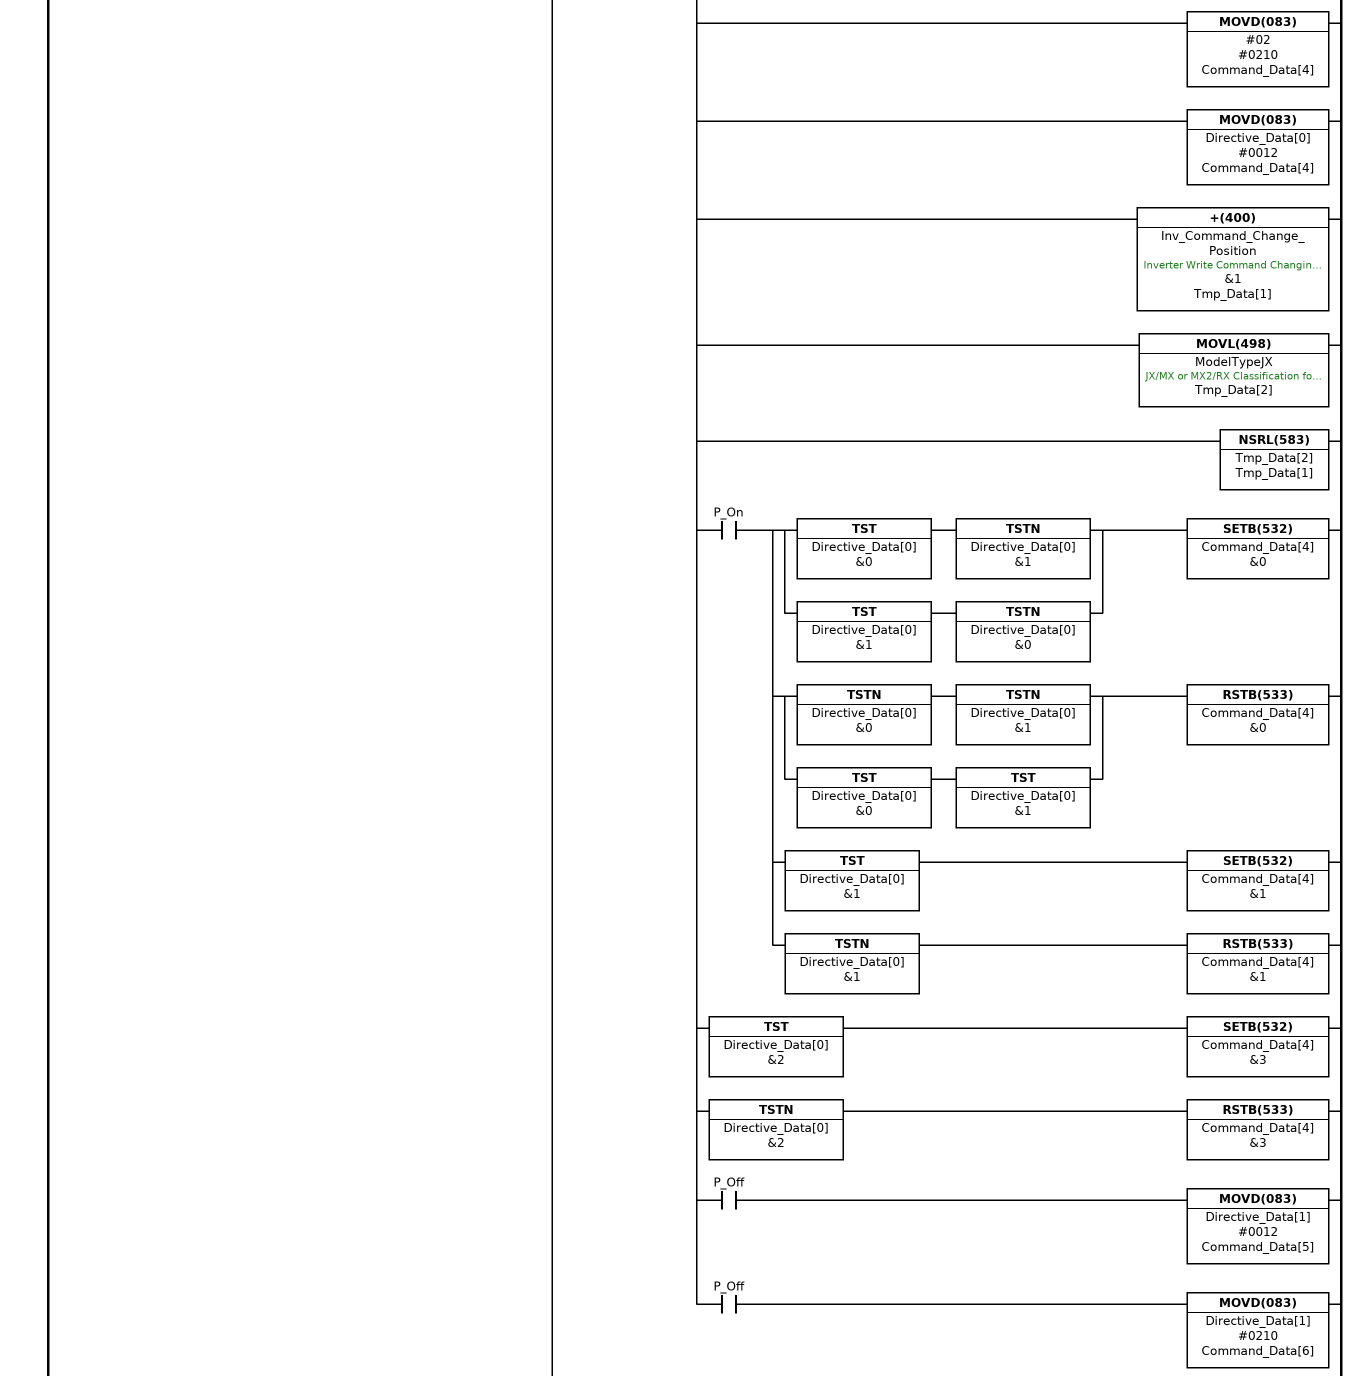

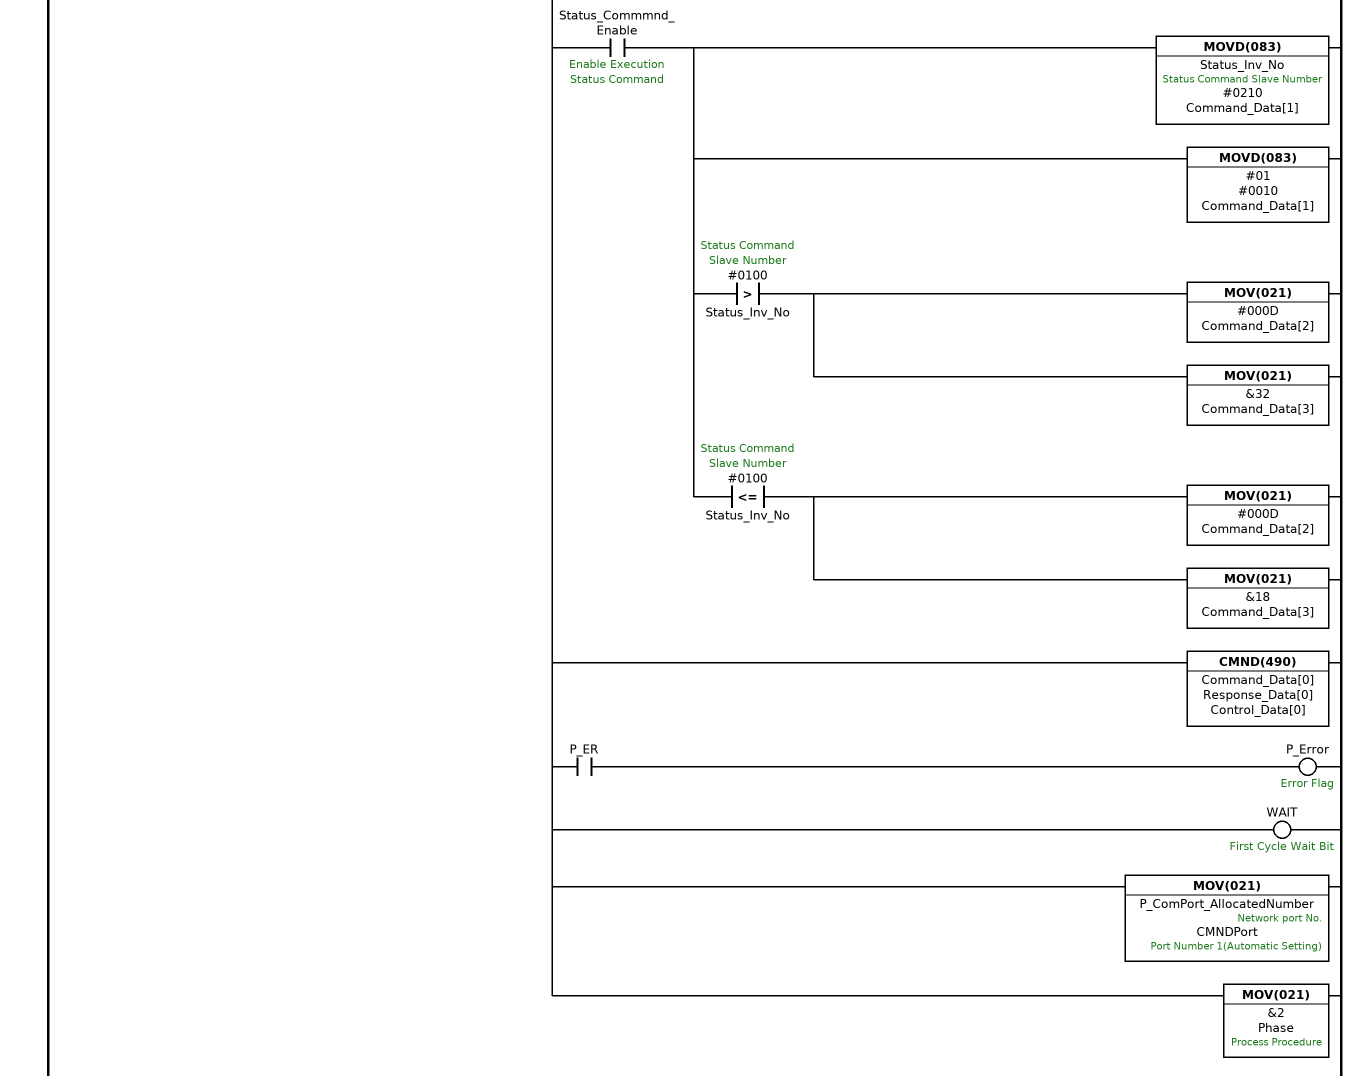
; rung 29: Execute CMND
LD AddressOk_Bit  ; Addrss Range Check OK Bit
AND BUSY_Run  ; Internal Processing Flag
AND P_ComPort_AutoAlloc_Available  ; Auto allocation avarable bit
AND=(300) &1 Phase  ; Process Procedure
OUT TR0
BSET(071) #0 Command_Data[0] Command_Data[21]
MOV(021) #2804 Command_Data[0]
AND Message_Command_Done  ; Exist Message Command Flag
XFER(070) &21 +24^IR1 Command_Data[1]
LD TR0
AND Command_Data_Change2
MOVD(083) Inv_Command_Change_Position #0210 Command_Data[1]  ; Inverter Write Command Changing Position
MOVD(083) #06 #0010 Command_Data[1]
MOV(021) #0001 Command_Data[2]
MOVD(083) Directive_Data[1] #0010 Command_Data[3]
MOVD(083) Directive_Data[1] #0212 Command_Data[3]
LD TR0
AND Command_Data_Change  ; Write Command Data Changing
OUT TR1
MOVD(083) Inv_Command_Change_Position #0210 Command_Data[1]  ; Inverter Write Command Changing Position
MOVD(083) #0F #0010 Command_Data[1]
MOV(021) #0000 Command_Data[2]
MOV(021) #0004 Command_Data[3]
MOVD(083) #02 #0210 Command_Data[4]
MOVD(083) Directive_Data[0] #0012 Command_Data[4]
+(400) Inv_Command_Change_Position &1 Tmp_Data[1]  ; Inverter Write Command Changing Position
MOVL(498) ModelTypeJX Tmp_Data[2]  ; JX/MX or MX2/RX Classification for older Inverter types also this Bit has to be set, like scanlist
NSRL(583) Tmp_Data[2] Tmp_Data[1]
AND P_On
OUT TR2
LDTST(350) Directive_Data[0] &0
ANDTSTN(351) Directive_Data[0] &1
LDTST(350) Directive_Data[0] &1
ANDTSTN(351) Directive_Data[0] &0
ORLD
ANDLD
SETB(532) Command_Data[4] &0
LD TR2
LDTSTN(351) Directive_Data[0] &0
ANDTSTN(351) Directive_Data[0] &1
LDTST(350) Directive_Data[0] &0
ANDTST(350) Directive_Data[0] &1
ORLD
ANDLD
RSTB(533) Command_Data[4] &0
LD TR2
ANDTST(350) Directive_Data[0] &1
SETB(532) Command_Data[4] &1
LD TR2
ANDTSTN(351) Directive_Data[0] &1
RSTB(533) Command_Data[4] &1
LD TR1
ANDTST(350) Directive_Data[0] &2
SETB(532) Command_Data[4] &3
LD TR1
ANDTSTN(351) Directive_Data[0] &2
RSTB(533) Command_Data[4] &3
LD TR1
AND P_Off
MOVD(083) Directive_Data[1] #0012 Command_Data[5]
LD TR1
AND P_Off
MOVD(083) Directive_Data[1] #0210 Command_Data[6]
LD TR0
AND Status_Commmnd_Enable  ; Enable Execution Status Command
OUT TR3
MOVD(083) Status_Inv_No #0210 Command_Data[1]  ; Status Command Slave Number
MOVD(083) #01 #0010 Command_Data[1]
AND>(320) #0100 Status_Inv_No  ; Status Command Slave Number
MOV(021) #000D Command_Data[2]
MOV(021) &32 Command_Data[3]
LD TR3
AND<=(315) #0100 Status_Inv_No  ; Status Command Slave Number
MOV(021) #000D Command_Data[2]
MOV(021) &18 Command_Data[3]
LD TR0
CMND(490) Command_Data[0] Response_Data[0] Control_Data[0]
AND P_ER
OUT P_Error  ; Error Flag
LD TR0
OUT WAIT  ; First Cycle Wait Bit
MOV(021) P_ComPort_AllocatedNumber CMNDPort  ; Network port No., Port Number 1(Automatic Setting)
MOV(021) &2 Phase  ; Process Procedure

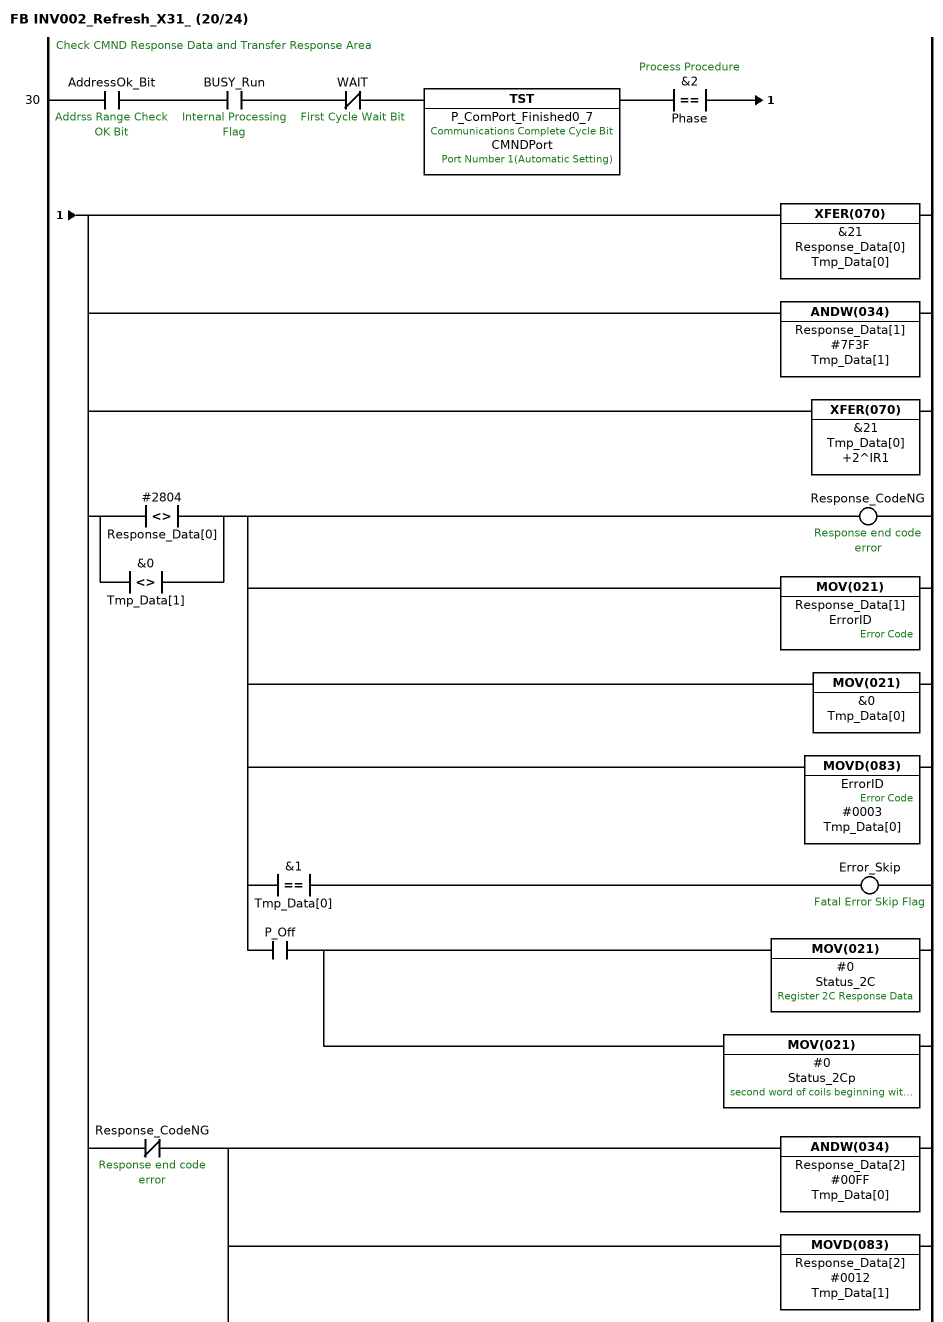

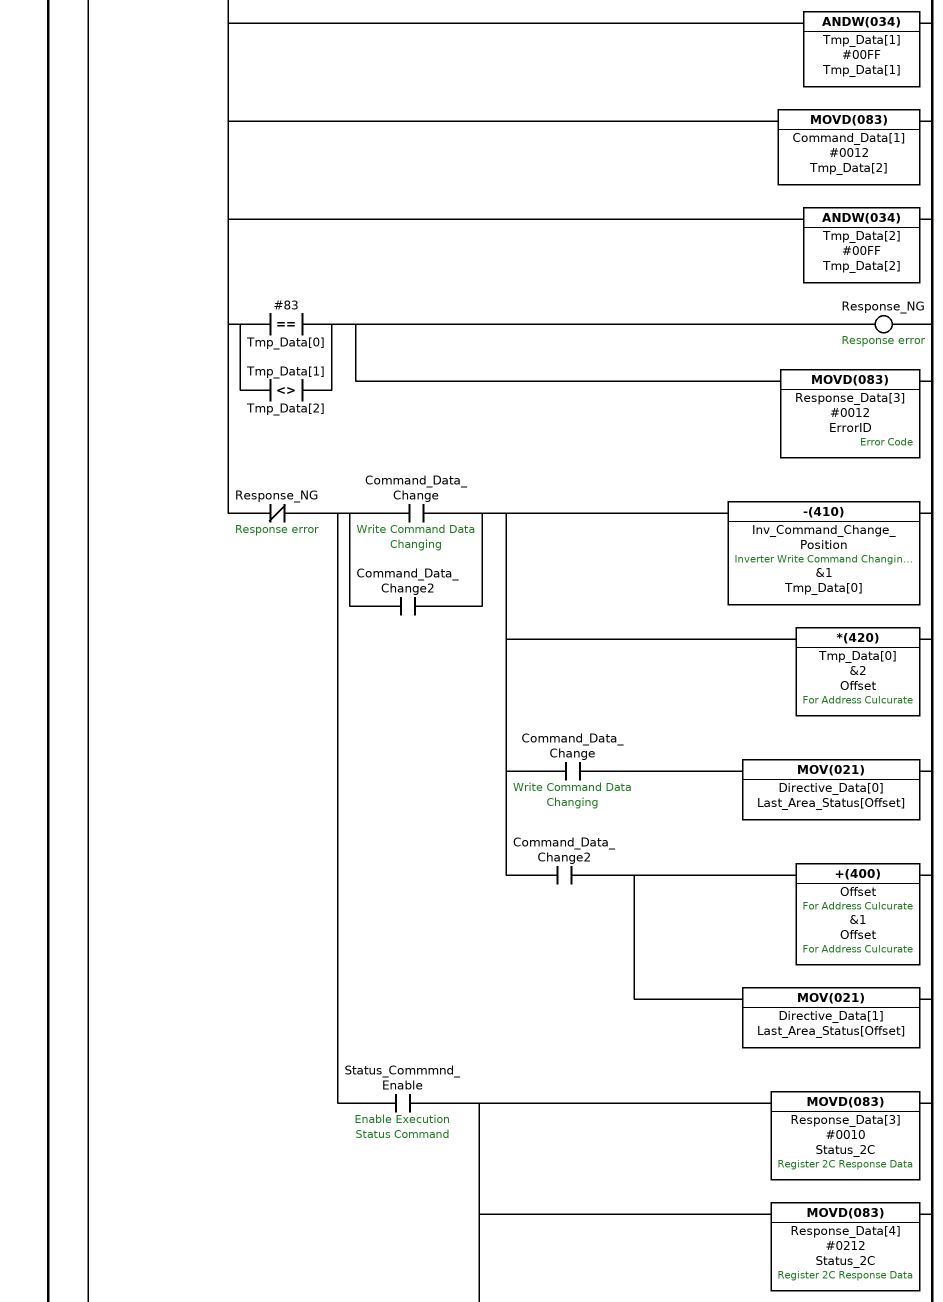

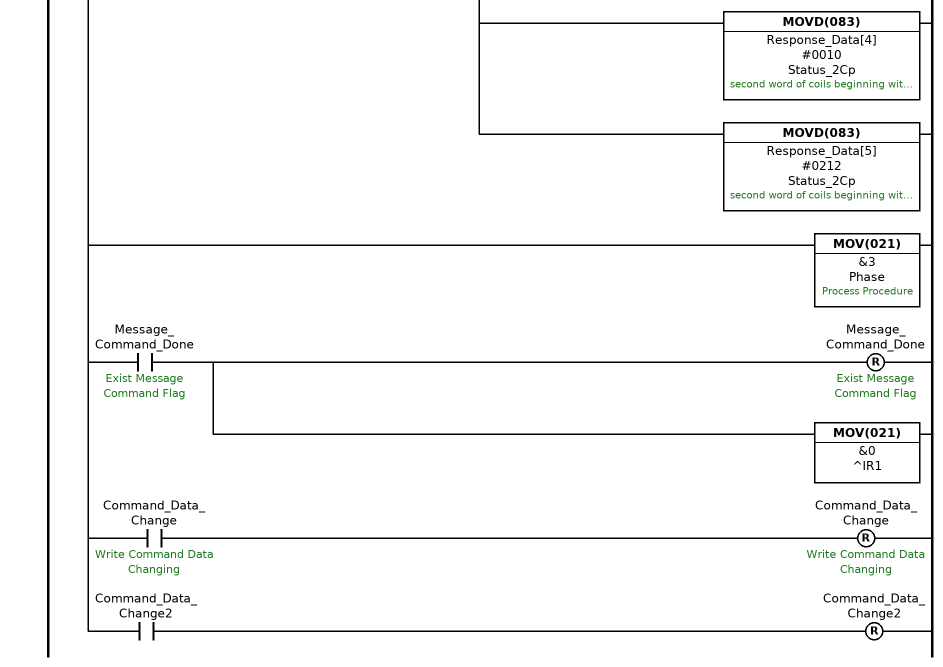
; rung 30: Check CMND Response Data and Transfer Response Area
LD AddressOk_Bit  ; Addrss Range Check OK Bit
AND BUSY_Run  ; Internal Processing Flag
ANDNOT WAIT  ; First Cycle Wait Bit
ANDTST(350) P_ComPort_Finished0_7 CMNDPort  ; Communications Complete Cycle Bit, Port Number 1(Automatic Setting)
AND=(300) &2 Phase  ; Process Procedure
OUT TR0
XFER(070) &21 Response_Data[0] Tmp_Data[0]
ANDW(034) Response_Data[1] #7F3F Tmp_Data[1]
XFER(070) &21 Tmp_Data[0] +2^IR1
LD<>(305) #2804 Response_Data[0]
OR<>(305) &0 Tmp_Data[1]
ANDLD
OUT TR1
OUT Response_CodeNG  ; Response end code error
MOV(021) Response_Data[1] ErrorID  ; Error Code
MOV(021) &0 Tmp_Data[0]
MOVD(083) ErrorID #0003 Tmp_Data[0]  ; Error Code
AND=(300) &1 Tmp_Data[0]
OUT Error_Skip  ; Fatal Error Skip Flag
LD TR1
AND P_Off
MOV(021) #0 Status_2C  ; Register 2C Response Data
MOV(021) #0 Status_2Cp  ; second word of coils beginning with coil 1F to 2E
LD TR0
ANDNOT Response_CodeNG  ; Response end code error
OUT TR2
ANDW(034) Response_Data[2] #00FF Tmp_Data[0]
MOVD(083) Response_Data[2] #0012 Tmp_Data[1]
ANDW(034) Tmp_Data[1] #00FF Tmp_Data[1]
MOVD(083) Command_Data[1] #0012 Tmp_Data[2]
ANDW(034) Tmp_Data[2] #00FF Tmp_Data[2]
LD=(300) #83 Tmp_Data[0]
OR<>(305) Tmp_Data[1] Tmp_Data[2]
ANDLD
OUT Response_NG  ; Response error
MOVD(083) Response_Data[3] #0012 ErrorID  ; Error Code
LD TR2
ANDNOT Response_NG  ; Response error
OUT TR3
LD Command_Data_Change  ; Write Command Data Changing
OR Command_Data_Change2
ANDLD
OUT TR4
-(410) Inv_Command_Change_Position &1 Tmp_Data[0]  ; Inverter Write Command Changing Position
*(420) Tmp_Data[0] &2 Offset  ; For Address Culcurate
AND Command_Data_Change  ; Write Command Data Changing
MOV(021) Directive_Data[0] Last_Area_Status[Offset]
LD TR4
AND Command_Data_Change2
+(400) Offset &1 Offset  ; For Address Culcurate
MOV(021) Directive_Data[1] Last_Area_Status[Offset]
LD TR3
AND Status_Commmnd_Enable  ; Enable Execution Status Command
MOVD(083) Response_Data[3] #0010 Status_2C  ; Register 2C Response Data
MOVD(083) Response_Data[4] #0212 Status_2C  ; Register 2C Response Data
MOVD(083) Response_Data[4] #0010 Status_2Cp  ; second word of coils beginning with coil 1F to 2E
MOVD(083) Response_Data[5] #0212 Status_2Cp  ; second word of coils beginning with coil 1F to 2E
LD TR0
MOV(021) &3 Phase  ; Process Procedure
AND Message_Command_Done  ; Exist Message Command Flag
RSET Message_Command_Done  ; Exist Message Command Flag
MOV(021) &0 ^IR1
LD TR0
AND Command_Data_Change  ; Write Command Data Changing
RSET Command_Data_Change  ; Write Command Data Changing
LD TR0
AND Command_Data_Change2
RSET Command_Data_Change2

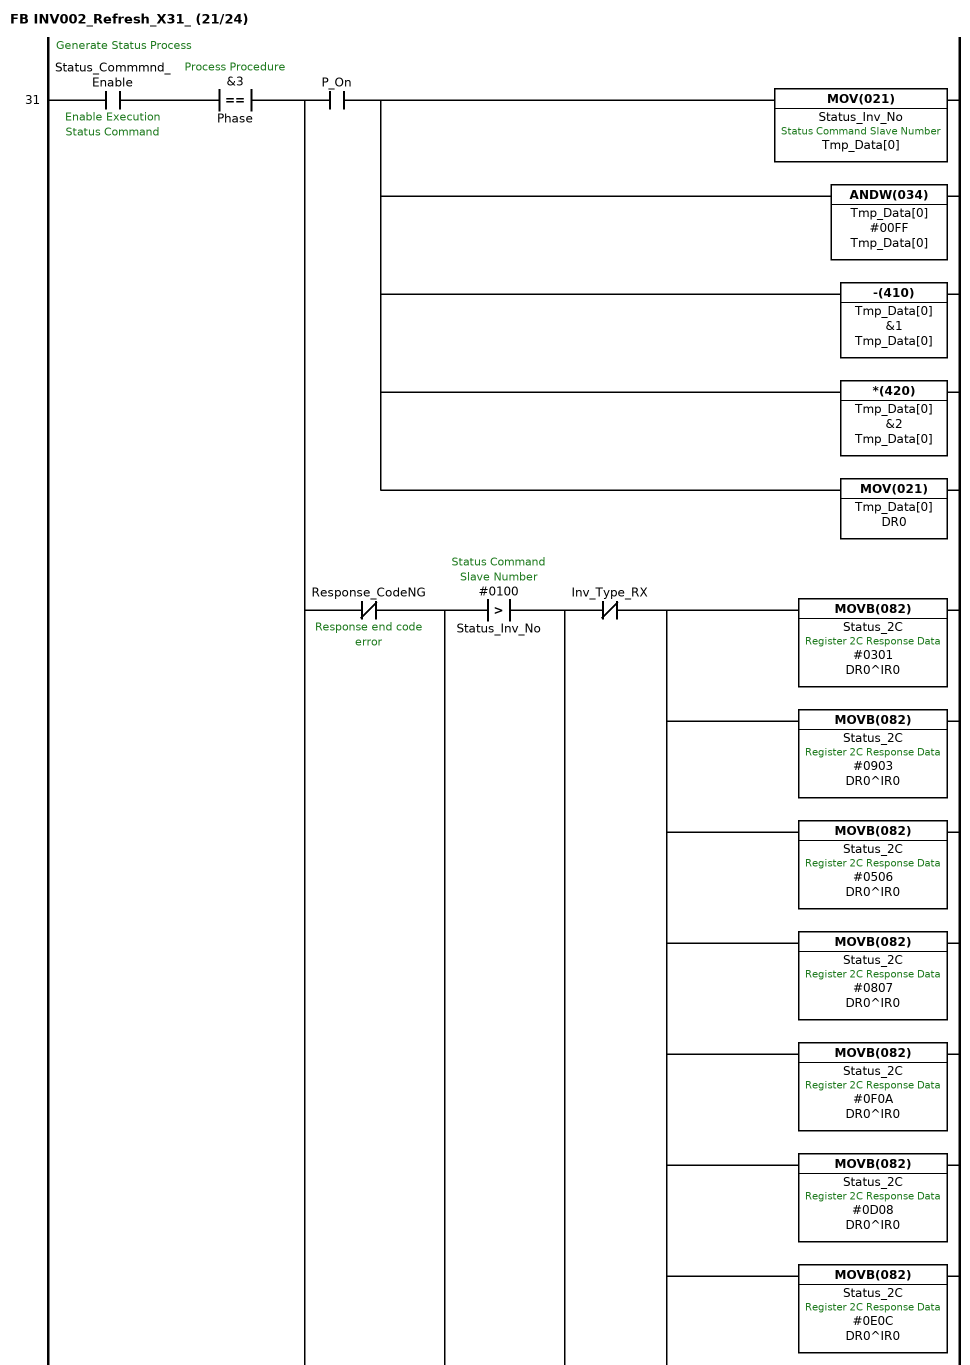

